sProdCodeAX5000 									:= 		F_ConvProductCodeToString(stSlaveIdentityAX5000);
//Get last 4 characters of the string
sProdCodeAX5000_End4 								:= 		RIGHT(sProdCodeAX5000, 4) ;
//Convert last 4 characters to a number
g_iHMI_ProdCodeAX5000 								:= 		STRING_TO_INT(sProdCodeAX5000_End4);

//In this function block the CRC counts for the individual counts can be decoded
fbAX5000_EcGetSlaveCrcErrorEx(	
							sNetId					:= 		gc_sADSNetID,
							nSlaveAddr				:= 		gc_uiAX5206_EtherCATAdr,
							bExecute				:= 		xExecute,
							tTimeout				:= 		T#2S,
							bBusy					=> 		xAX5000GetSlaveCrc_Busy,
							bError					=> 		xAX5000GetSlaveCrc_Error,
							nErrId					=> 		udiAX5000GetSlaveCrc_ErrId,
							crcError				=> 		g_stHMI_AX5000CrcErrorEx );

//Working Counter: Should remain Zero, If value=1 then data is bad from this device
g_xAX5000_Wc ;


//Get the STATE of the AX5805 terminal and display as a text string
g_sHMI_StateAX5805 									:= 		F_ConvStateToString(g_wStateAX5805);

// slave device's STATE BITS  
g_stHMI_AX5805EcSlaveStateBits 						:=  	F_ConvSlaveStateToBits(g_stAX5805EcSlaveState);

fbAX5805_EcGetSlaveIdentity(		
							sNetId					:= 		gc_sADSNetID,
							nSlaveAddr				:= 		gc_uiAX5805_EtherCATAdr,
							bExecute				:= 		xExecute,
							tTimeout				:= 		T#2S,
							bBusy					=> 		xAX5805SlaveIdentity_Busy,
							bError					=> 		xAX5805SlaveIdentity_Error,
							nErrId					=> 		udiAX5805SlaveIdentity_ErrId,
							identity				=> 		stSlaveIdentityAX5805 );

sProdCodeAX5805 									:= 		F_ConvProductCodeToString(stSlaveIdentityAX5805);
//Get last 4 characters of the string
sProdCodeAX5805_End4 								:= 		RIGHT(sProdCodeAX5805, 4) ;
//Convert last 4 characters to a number
g_iHMI_ProdCodeAX5805 								:= 		STRING_TO_INT(sProdCodeAX5805_End4);

//In this function block the CRC counts for the individual counts can be decoded
fbAX5805_EcGetSlaveCrcErrorEx(	
							sNetId					:= 		gc_sADSNetID,
							nSlaveAddr				:= 		gc_uiAX5805_EtherCATAdr,
							bExecute				:= 		xExecute,
							tTimeout				:= 		T#2S,
							bBusy					=> 		xAX5805GetSlaveCrc_Busy,
							bError					=> 		xAX5805GetSlaveCrc_Error,
							nErrId					=> 		udiAX5805GetSlaveCrc_ErrId,
							crcError				=> 		g_stHMI_AX5805CrcErrorEx );

//Working Counter: Should remain Zero, If value=1 then data is bad from this device
g_xAX5805_Wc ;


//Get the STATE of the EP1908-0002 module and display as a text string
g_sHMI_StateEP1908 									:= 		F_ConvStateToString(g_wStateEP1908);

// slave device's STATE BITS  
g_stHMI_EP1908EcSlaveStateBits 						:=  	F_ConvSlaveStateToBits(g_stEP1908EcSlaveState);

fbEP1908_EcGetSlaveIdentity(		
							sNetId					:= 		gc_sADSNetID,
							nSlaveAddr				:= 		gc_uiEP1908_EtherCATAdr,
							bExecute				:= 		xExecute,
							tTimeout				:= 		T#2S,
							bBusy					=> 		xEP1908SlaveIdentity_Busy,
							bError					=> 		xEP1908SlaveIdentity_Error,
							nErrId					=> 		udiEP1908SlaveIdentity_ErrId,
							identity				=> 		stSlaveIdentityEP1908 );

sProdCodeEP1908 									:= 		F_ConvProductCodeToString(stSlaveIdentityEP1908);
//Get last 4 characters of the string
sProdCodeEP1908_End4 								:= 		RIGHT(sProdCodeEP1908, 4) ;
//Convert last 4 characters to a number
g_iHMI_ProdCodeEP1908 								:= 		STRING_TO_INT(sProdCodeEP1908_End4);

//In this function block the CRC counts for the individual counts can be decoded
fbEP1908_EcGetSlaveCrcErrorEx(	
							sNetId					:= 		gc_sADSNetID,
							nSlaveAddr				:= 		gc_uiEP1908_EtherCATAdr,
							bExecute				:= 		xExecute,
							tTimeout				:= 		T#2S,
							bBusy					=> 		xEP1908GetSlaveCrc_Busy,
							bError					=> 		xEP1908GetSlaveCrc_Error,
							nErrId					=> 		udiEP1908GetSlaveCrc_ErrId,
							crcError				=> 		g_stHMI_EP1908CrcErrorEx );

//Working Counter: Should remain Zero, If value=1 then data is bad from this device
g_xEP1908_Wc ;

*)

//END_IF ;

END_PROGRAM

// ---- POUs/Control_System_Diagnostics/System_Functions.TcPOU
PROGRAM System_Functions
//		8-2-2012
// 		This Program has been supplied by Beckhoff Automation As-Is and is intended only as an example 
//		implementation. Functionality is not guaranteed. 
//
VAR
	//General timer for periodic reads
	T1									:		TON ;
	xExecute							:		BOOL ;
	tTime1								:		TIME ;

	//Get Device Identification
	fbGetDeviceIdentificationEx			:		FB_GetDeviceIdentificationEx ;
	xGetDeviceId_Busy					:		BOOL ;
	xGetDeviceId_Error					:		BOOL ;
	udiGetDeviceId_ErrId				:		UDINT ;
	stDevIdent							:		ST_DeviceIdentificationEx ;

	//Get ADS Router Info
	fbGetRouterStatusInfo				:		FB_GetRouterStatusInfo ;
	xGetRouterStatusInfo_Busy			:		BOOL ;
	xGetRouterStatusInfo_Error			:		BOOL ;
	udiGetRouterStatusInfo_ErrId		:		UDINT ;
	stRouterStatusInfo					:		ST_TcRouterStatusInfo ;


(*
(* Get CPU Usage Info  *)
	fbTC_CpuUsage: TC_CpuUsage;
	bCpuUsage_Busy: BOOL;
	bCpuUsage_Error: BOOL;
	nCpuUsage_ErrId: UDINT;
	nCpuUsage: UDINT;
	nCpuUsage_HMI: UDINT;

(* Get System Latency Values *)
	fbTC_SysLatency: TC_SysLatency;
	bSysLatency_Busy: BOOL;
	bSysLatency_Error: BOOL;
	nSysLatency_ErrId: UDINT;
	nSysLatency_Actual: UDINT;
	nSysLatency_Max: UDINT;
	nSysLatency_Actual_HMI: UDINT;
	nSysLatency_Max_HMI: UDINT;

(* SystemTaskInfoArr[1].cycleTime is in 100ns increments - needed to convert to ms for display*)
	nCycleTime_HMI: LREAL;

(* SystemTaskInfoArr[1].lastExecTime is in 100ns increments - needed to convert to ms for display*)
	nLastExecTime_HMI: LREAL;
	fbGetDeviceIdentificationEx: FB_GetDeviceIdentificationEx;
*)
	fbFB_MDP_ScanModules				: 		FB_MDP_ScanModules;
	eMDP_ModType						: 		E_MDP_ModuleType;
	usiModIdx							: 		USINT;
	xMDP_ScanModules_busy				: 		BOOL;
	xMDP_ScanModules_Error				: 		BOOL;
	udiMDP_ScanModules_ErrID			: 		UDINT;
	bMDP_ScanModules_DynModID			: 		BYTE;
	usiMDP_ScanModules_ModTypCnt		: 		USINT;
	usiMDP_ScanModules_ModCnt			: 		USINT;

	fbFB_MDP_ReadModuleContent 			:		FB_MDP_ReadModuleContent ;
	ST_MDP_Addr 						:		ST_MDP_Addr ;
	dwMB_Buffer							: 		DWORD ;
	xMDP_Motherboard_ReadModContent_Busy: 		BOOL ;
	xMDP_Motherboard_ReadModContent_Error: 		BOOL ;
	udiMDP_Motherboard_ReadModContent_ErrID: 	UDINT ;
	usiMDP_Motherboard_ReadModContent_ErrPOS: 	USINT ;
	arrMDP_Motherboard_StartIdx			: 		ARRAY [0..255] OF UINT ;

	fbFB_MDP_SplitErrorID				: 		FB_MDP_SplitErrorID ;
	eMDP_ErrGroup 						:		E_MDP_ErrGroup ;
	uiMDP_Motherboard_ReadModContent_ErrCODE:	UINT ;

	fbFB_MDP_ReadModuleHeader			: 		FB_MDP_ReadModuleHeader ;
	xMDP_Motherboard_ReadModHeader_Busy	: 		BOOL ;
	xMDP_Motherboard_ReadModHeader_Error: 		BOOL ;
	udiMDP_Motherboard_ReadModHeader_ErrID: 	UDINT ;
	ST_MDP_Motherboard_ReadModHeader 	:		ST_MDP_ModuleHeader ;

	fbFB_MDP_CPU_Read1					: 		FB_MDP_CPU_Read;
	ST_CPUModHdr 						:		ST_MDP_ModuleHeader ;
	ST_CPUModContent 					: 		ST_MDP_CPU ;

	fbFB_MDP_Mainboard_ReadTBL1			: 		FB_MDP_Mainboard_ReadTBL1;
	ST_MainboardModHdrTBL1				:		ST_MDP_ModuleHeader ;
	ST_MainboardModContentTBL1			: 		ST_MDP_MainboardTBL1 ;

	fbFB_MDP_Mainboard_ReadTBL2			: 		FB_MDP_Mainboard_ReadTBL2 ;
	ST_MainboardModHdrTBL2				:		ST_MDP_ModuleHeader ;
	ST_MainboardModContentTBL2			: 		ST_MDP_MainboardTBL2 ;

	fbFB_MDP_Mainboard_ReadTBL3			: 		FB_MDP_Mainboard_ReadTBL3 ;
	ST_MainboardModHdrTBL3				:		ST_MDP_ModuleHeader ;
	ST_MainboardModContentTBL3			: 		ST_MDP_MainboardTBL3 ;

	fbFB_MDP_Mainboard_ReadTBL4			: 		FB_MDP_Mainboard_ReadTBL4 ;
	ST_MainboardModHdrTBL4				:		ST_MDP_ModuleHeader ;
	ST_MainboardModContentTBL4			: 		ST_MDP_MainboardTBL4 ;
	
	fbFB_MDP_NIC0_Read					: 		FB_MDP_NIC_Read ;
	ST_NIC0_ModHdr						: 		ST_MDP_ModuleHeader ;
	ST_NIC0_ModContent					: 		ST_MDP_NIC_Properties ;
	
	fbFB_MDP_NIC1_Read					: 		FB_MDP_NIC_Read ;
	ST_NIC1_ModHdr						: 		ST_MDP_ModuleHeader ;
	ST_NIC1_ModContent					: 		ST_MDP_NIC_Properties ;	
	lrOperTimeHrs						: 		LREAL ;
	lrOperTimeDays						: 		LREAL ;
	lrOperTimeYears						: 		LREAL ;

	fbFB_MDP_Time1_Read					: 		FB_MDP_Time_ReadTBL1 ;
	ST_Time1_ModHdr						: 		ST_MDP_ModuleHeader ;
	ST_Time1_ModContent					: 		ST_MDP_TimeTBL1 ;
END_VAR

//		8-2-2012
// 		This Program has been supplied by Beckhoff Automation As-Is and is intended only as an example 
//		implementation. Functionality is not guaranteed. 
//

//IF g_bHMI_ScreenBeingDisplayed = 90 THEN
//Create the xExecute bit for continuous timed interval FB calls
T1(IN:= NOT xExecute, PT:= T#2S, Q=> xExecute, ET=>tTime1 );

(* Computer/Controller Device Info - Get CX and TwinCAT version info
   from the resulting structure "stDevIdent" - display only when the 
   function block is not BUSY retrieving the data else the display
   will "blink" because while the FB is BUSY the values go to 0 or
   "blank" text *)
fbGetDeviceIdentificationEx(
							bExecute					:= 		xExecute, 
							tTimeout					:= 		T#2S, 
							sNetId						:= 		'', 
							bBusy						=> 		xGetDeviceId_Busy, 
							bError						=> 		xGetDeviceId_Error, 
							nErrorID					=> 		udiGetDeviceId_ErrId, 
							stDevIdent					=> 		stDevIdent );
							
IF NOT xGetDeviceId_Busy THEN 
							g_stHMI_DevIdent 			:= 		stDevIdent ; 
END_IF ;

g_stHMI_AppInfo 										:= _AppInfo  ;

//ADS Router Status info
fbGetRouterStatusInfo(		
							sNetId						:= 		'',
							bExecute					:= 		xExecute,
							tTimeout					:= 		T#2S,
							bBusy						=> 		xGetRouterStatusInfo_Busy,
							bError						=> 		xGetRouterStatusInfo_Error,
							nErrID						=> 		udiGetRouterStatusInfo_ErrId,
							info						=> 		stRouterStatusInfo );
							
IF NOT xGetRouterStatusInfo_Busy THEN 
							g_stHMI_RouterStatusInfo	:= 		stRouterStatusInfo ; 
END_IF ;

g_stHMI_PlcTaskSystemInfo 								:= 		_TaskInfo[_AppInfo.TaskCnt] ;
g_lrHMI_PlcTaskSystemInfo_CycleTime 					:= 		g_stHMI_PlcTaskSystemInfo.CycleTime / 10.0 ;
g_lrHMI_PlcTaskSystemInfo_LastExecTime 					:= 		g_stHMI_PlcTaskSystemInfo.LastExecTime / 10.0 ;

//In order to be able to query or set an MDP parameter, the Dynamic Module ID of 
//the module in which the parameter is located must be known.
fbFB_MDP_ScanModules(
							bExecute					:= 		xExecute, 
							nModuleType					:= 		eMDP_ModType, 
							iModIdx						:= 		usiModIdx, 
							tTimeout					:= 		T#2S, 
							sAmsNetId					:= 		'', 
							bBusy						=> 		xMDP_ScanModules_busy, 
							bError						=> 		xMDP_ScanModules_Error, 
							nErrID						=> 		udiMDP_ScanModules_ErrID, 
							nDynModuleId				=> 		bMDP_ScanModules_DynModID, 
							iModuleTypeCount			=> 		usiMDP_ScanModules_ModTypCnt, 
							iModuleCount				=> 		usiMDP_ScanModules_ModCnt );

// The function block enables the header of an MDP module to be queried
fbFB_MDP_ReadModuleHeader(
							bExecute					:= 		xExecute, 
							nDynModuleId				:= 		4, 
							tTimeout					:= 		T#2S, 
							sAmsNetId					:= 		'', 
							bBusy						=> 		xMDP_Motherboard_ReadModHeader_Busy, 
							bError						=> 		xMDP_Motherboard_ReadModHeader_Error, 
							nErrID						=> 		udiMDP_Motherboard_ReadModHeader_ErrID, 
							stMDP_ModHeader				=> 		ST_MDP_Motherboard_ReadModHeader);							
							

fbFB_MDP_CPU_Read1(
							xExecute					:= 		xExecute, 
							tTimeout					:= 		T#2S, 
							usiModIdx					:= 		0, 
							sAmsNetId					:= 		'', 
							bBusy						=> 		, 
							bError						=> 		, 
							nErrID						=> 		, 
							iErrPos						=> 		, 
							stMDP_ModuleHeader			=> 		ST_CPUModHdr, 
							stMDP_ModuleContent			=> 		ST_CPUModContent);							

g_lrHMI_CPUfrequency 									:=		ST_CPUModContent.udiCPUfrequency / 1000.0	; // CPU Clock Frequency in GHz				
g_iHMI_CPUusage											:=		ST_CPUModContent.uiCPUusage ;  // CPU Usage in percent
g_iHMI_CPUtemperature 									:= 		ST_CPUModContent.iCPUtemp ; // CPU Temperature in DegC	

fbFB_MDP_Mainboard_ReadTBL1(
							xExecute					:= 		xExecute, 
							tTimeout					:= 		T#2S, 
							usiModIdx					:= 		0, 
							sAmsNetId					:= 		'', 
							bBusy						=> 		, 
							bError						=> 		, 
							nErrID						=> 		, 
							iErrPos						=> 		, 
							stMDP_ModuleHeader			=> 		ST_MainboardModHdrTBL1, 
							stMDP_ModuleContent			=> 		ST_MainboardModContentTBL1);


g_sHMI_MainboardType 									:= 		ST_MainboardModContentTBL1.sMainboardType ;
g_sHMI_MainboardSN 										:= 		ST_MainboardModContentTBL1.sMainboardSN ;
g_sHMI_MainboardProdDate								:= 		ST_MainboardModContentTBL1.sMainboardProdDate ;
g_udiHMI_MainboardBootCount								:= 		ST_MainboardModContentTBL1.udiMainboardBootCount ;
lrOperTimeHrs											:= 		ST_MainboardModContentTBL1.udiMainboardOperTime / 60.0 ;
lrOperTimeDays											:= 		lrOperTimeHrs / 24.0 ;
g_udiHMI_MainboardOperTimeDays 							:= 		TRUNC(lrOperTimeDays) ;
g_lrHMI_MainboardOperTimeHrs							:=		24.0 * (lrOperTimeDays - UDINT_TO_LREAL(g_udiHMI_MainboardOperTimeDays)) ;
g_diHMI_MainboardMinTemp								:= 		ST_MainboardModContentTBL1.diMainboardMinTemp ;
g_diHMI_MainboardMaxTemp								:= 		ST_MainboardModContentTBL1.diMainboardMaxTemp ;
g_lrHMI_MainboardMinVolt								:= 		ST_MainboardModContentTBL1.diMainboardMinVolt / 1000.0 ;
g_lrHMI_MainboardMaxVolt								:= 		ST_MainboardModContentTBL1.diMainboardMaxVolt / 1000.0 ;
g_iHMI_MainboardActualTemp								:= 		ST_MainboardModContentTBL1.iMainboardActualTemp ;


fbFB_MDP_Mainboard_ReadTBL2(
							xExecute					:= 		xExecute, 
							tTimeout					:= 		T#2S, 
							usiModIdx						:= 		0, 
							sAmsNetId					:= 		'', 
							bBusy						=> 		, 
							bError						=> 		, 
							nErrID						=> 		, 
							iErrPos						=> 		, 
							stMDP_ModuleHeader			=> 		ST_MainboardModHdrTBL2, 
							stMDP_ModuleContent			=> 		ST_MainboardModContentTBL2);


g_bHMI_MainboardRevision 								:= 		ST_MainboardModContentTBL2.usiMainboardRevision ;
g_bHMI_MainboardBiosMajVers 							:= 		ST_MainboardModContentTBL2.usiMainboardBiosMajVers ;
g_bHMI_MainboardBiosMinVers 							:= 		ST_MainboardModContentTBL2.usiMainboardBiosMinVers ;


fbFB_MDP_Mainboard_ReadTBL3(
							xExecute					:= 		xExecute, 
							tTimeout					:= 		T#2S, 
							usiModIdx						:= 		0, 
							sAmsNetId					:= 		'', 
							bBusy						=> 		, 
							bError						=> 		, 
							nErrID						=> 		, 
							iErrPos						=> 		, 
							stMDP_ModuleHeader			=> 		ST_MainboardModHdrTBL3, 
							stMDP_ModuleContent			=> 		ST_MainboardModContentTBL3);							

g_sHMI_Mainboard1p05v 									:= 		ST_MainboardModContentTBL3.sMainboard1p05v ;
g_sHMI_MainboardVccCore 								:= 		ST_MainboardModContentTBL3.sMainboardVccCore ;
g_sHMI_Mainboard5v 										:= 		ST_MainboardModContentTBL3.sMainboard5v ;
g_sHMI_Mainboard12v 									:= 		ST_MainboardModContentTBL3.sMainboard12v ;
g_sHMI_MainboardVBatt 									:= 		ST_MainboardModContentTBL3.sMainboardVBatt ;
g_sHMI_MainboardPwrCtrlVcc 								:= 		ST_MainboardModContentTBL3.sMainboardPwrCtrlVcc ;
g_sHMI_MainboardCX2100_5v 								:= 		ST_MainboardModContentTBL3.sMainboardCX2100_5v ;
g_sHMI_MainboardCX2100_12v 								:= 		ST_MainboardModContentTBL3.sMainboardCX2100_12v ;
g_sHMI_MainboardCX2100_24v 								:= 		ST_MainboardModContentTBL3.sMainboardCX2100_24v ;

					
fbFB_MDP_Mainboard_ReadTBL4(
							xExecute					:= 		xExecute, 
							tTimeout					:= 		T#2S, 
							usiModIdx						:= 		0, 
							sAmsNetId					:= 		'', 
							bBusy						=> 		, 
							bError						=> 		, 
							nErrID						=> 		, 
							iErrPos						=> 		, 
							stMDP_ModuleHeader			=> 		ST_MainboardModHdrTBL4, 
							stMDP_ModuleContent			=> 		ST_MainboardModContentTBL4);

g_lrHMI_Mainboard1p05v 									:= 		ST_MainboardModContentTBL4.iMainboard1p05v / 1000.0 ;
g_lrHMI_MainboardVccCore 								:= 		ST_MainboardModContentTBL4.iMainboardVccCore / 1000.0 ;
g_lrHMI_Mainboard5v 									:= 		ST_MainboardModContentTBL4.iMainboard5v / 1000.0 ;
g_lrHMI_Mainboard12v 									:= 		ST_MainboardModContentTBL4.iMainboard12v / 1000.0 ;
g_lrHMI_MainboardVBatt 									:= 		ST_MainboardModContentTBL4.iMainboardVBatt / 1000.0 ;
g_lrHMI_MainboardPwrCtrlVcc 							:= 		ST_MainboardModContentTBL4.iMainboardPwrCtrlVcc / 1000.0 ;
g_lrHMI_MainboardCX2100_5v 								:= 		ST_MainboardModContentTBL4.iMainboardCX2100_5v / 1000.0 ;
g_lrHMI_MainboardCX2100_12v 							:= 		ST_MainboardModContentTBL4.iMainboardCX2100_12v / 1000.0 ;
g_lrHMI_MainboardCX2100_24v 							:= 		ST_MainboardModContentTBL4.iMainboardCX2100_24v / 1000.0 ; 


fbFB_MDP_NIC0_Read(
							xExecute					:= 		xExecute, 
							tTimeout					:= 		T#2S, 
							usiModIdx					:= 		0, 
							sAmsNetId					:= 		'', 
							bBusy						=> 		, 
							bError						=> 		, 
							nErrID						=> 		, 
							iErrPos						=> 		, 
							stMDP_ModuleHeader			=> 		ST_NIC0_ModHdr, 
							stMDP_ModuleContent			=> 		ST_NIC0_ModContent);

fbFB_MDP_NIC1_Read(
							xExecute					:= 		xExecute, 
							tTimeout					:= 		T#2S, 
							usiModIdx					:= 		1, 
							sAmsNetId					:= 		'', 
							bBusy						=> 		, 
							bError						=> 		, 
							nErrID						=> 		, 
							iErrPos						=> 		, 
							stMDP_ModuleHeader			=> 		ST_NIC1_ModHdr, 
							stMDP_ModuleContent			=> 		ST_NIC1_ModContent);

fbFB_MDP_Time1_Read(
							xExecute					:= 		xExecute, 
							tTimeout					:= 		T#2S, 
							usiModIdx					:= 		0, 
							sAmsNetId					:= 		'', 
							bBusy						=> 		, 
							bError						=> 		, 
							nErrID						=> 		, 
							iErrPos						=> 		, 
							stMDP_ModuleHeader			=> 		ST_Time1_ModHdr, 
							stMDP_ModuleContent			=> 		ST_Time1_ModContent);				
//	END_IF ;

END_PROGRAM

// ---- POUs/MDP_Function_Blocks/FB_MDP_Mainboard_ReadTBL1.TcPOU
FUNCTION_BLOCK FB_MDP_Mainboard_ReadTBL1

VAR_INPUT
	xExecute				: BOOL;								// Function block execution is triggered by a rising edge at this input
	tTimeout				: TIME		:= DEFAULT_ADS_TIMEOUT;	// States the time before the function is cancelled
	usiModIdx				: USINT		:= 0;					// Index number of chosen MDP device
	sAmsNetId				: T_AmsNetId;						// keep empty '' for the local device
END_VAR

VAR_OUTPUT
	xBusy					: BOOL;
	xError					: BOOL;
	udiErrID				: UDINT;
	usiErrPos				: USINT;							// If a subindex is not supported, iErrPos indicates at which subindex the error appears first
	stMDP_ModuleHeader		: ST_MDP_ModuleHeader;
	stMDP_ModuleContent		: ST_MDP_MainboardTBL1;	
END_VAR

VAR
	fbMDP_ReadModule		: FB_MDP_ReadModule;
	arrData					: ARRAY[0..60] OF BYTE;				// requested data
	arrStartIdx				: ARRAY[0..15] OF UINT;				// startindexes in bytes of each subindex element

	stMDP_Addr				: ST_MDP_Addr;
	eModuleType				: E_MDP_ModuleType;
	usiSubIdxCount			: USINT;

	xSubExecute				: BOOL;
	xReadBusy				: BOOL;

	RisingEdge				: R_TRIG;
	TimeOut					: TON;								// general timeout	
END_VAR

RisingEdge( CLK					:= xExecute );
IF NOT xBusy THEN										// FB only react to the external execute if it is not busy
	IF RisingEdge.Q THEN
		xBusy					:= TRUE;

		// reset variables
		xError					:= FALSE;
		udiErrID				:= 0;
		usiErrPos				:= 0;
		xSubExecute				:= TRUE;

		// specific values for Mainboard content
		stMDP_Addr.nArea		:= 16#08;
//		stMDP_Addr.nModuleId;							will be allocated dynamically
		stMDP_Addr.nTableId		:= 16#01;
//		stMDP_Addr.nFlag;								not used up to now
//		stMDP_Addr.nSubIdx;								all subindexes will be requested
		eModuleType				:= eMDP_ModT_Mainboard;
		usiSubIdxCount			:= 11;					// TableId 16#01 contains 10 elements

		MEMSET( ADR(arrData), 0, SIZEOF(arrData) );		// reset buffer

		TimeOut(IN 				:= FALSE);
		TimeOut(PT 				:= tTimeout, IN 	:= TRUE);
	END_IF
END_IF


IF xBusy THEN
	IF xSubExecute THEN
		xSubExecute 			:= FALSE;

		fbMDP_ReadModule( bExecute := FALSE );
		fbMDP_ReadModule(
			stMDP_Addr			:= stMDP_Addr,
			eModuleType			:= eModuleType,
			iModIdx				:= usiModIdx,
			iSubIdxCount		:= usiSubIdxCount,
			bExecute			:= TRUE,
			tTimeout			:= tTimeout,
			pDstBuf				:= ADR(arrData),
			cbDstBufLen			:= SIZEOF(arrData),
			sAmsNetId			:= sAmsNetId,

			bBusy				=> xReadBusy,
			bError				=> xError,
			nErrID				=> udiErrID,
			iErrPos				=> usiErrPos,
			stMDP_DynAddr		=> ,
			iModuleTypeCount	=> ,
			iModuleCount		=> ,
			stMDP_ModuleHeader	=> ,
			arrStartIdx			=> ,
		);
	ELSE
		fbMDP_ReadModule(
			bExecute			:= FALSE,

			bBusy				=> xReadBusy,
			bError				=> xError,
			nErrID 				=> udiErrID,
			iErrPos				=> usiErrPos,
		 );
		IF NOT xReadBusy THEN
			// allocate received module header
			stMDP_ModuleHeader	:= fbMDP_ReadModule.stMDP_ModuleHeader;
			// allocate information of startindexes in data buffer
			MEMCPY(ADR(arrStartIdx), ADR(fbMDP_ReadModule.arrStartIdx), SIZEOF(arrStartIdx) );
			// reset module content struct
			MEMSET( ADR(stMDP_ModuleContent), 0, SIZEOF(stMDP_ModuleContent) );
			// allocate received data to NIC struct
			stMDP_ModuleContent.uiLen		:= arrData[0];
			MEMCPY(ADR(stMDP_ModuleContent.sMainboardType),			ADR(arrData)+arrStartIdx[1],	MIN(arrStartIdx[2]-arrStartIdx[1],	SIZEOF(stMDP_ModuleContent.sMainboardType))     );
			MEMCPY(ADR(stMDP_ModuleContent.sMainboardSN),			ADR(arrData)+arrStartIdx[2],	MIN(arrStartIdx[3]-arrStartIdx[2],	SIZEOF(stMDP_ModuleContent.sMainboardSN))     );
			MEMCPY(ADR(stMDP_ModuleContent.sMainboardProdDate),		ADR(arrData)+arrStartIdx[3],	MIN(arrStartIdx[4]-arrStartIdx[3],	SIZEOF(stMDP_ModuleContent.sMainboardProdDate))     );
			MEMCPY(ADR(stMDP_ModuleContent.udiMainboardBootCount),	ADR(arrData)+arrStartIdx[4],	MIN(arrStartIdx[5]-arrStartIdx[4],	SIZEOF(stMDP_ModuleContent.udiMainboardBootCount))     );
			MEMCPY(ADR(stMDP_ModuleContent.udiMainboardOperTime),	ADR(arrData)+arrStartIdx[5],	MIN(arrStartIdx[6]-arrStartIdx[5],	SIZEOF(stMDP_ModuleContent.udiMainboardOperTime))     );
			MEMCPY(ADR(stMDP_ModuleContent.diMainboardMinTemp),		ADR(arrData)+arrStartIdx[6],	MIN(arrStartIdx[7]-arrStartIdx[6],	SIZEOF(stMDP_ModuleContent.diMainboardMinTemp))     );
			MEMCPY(ADR(stMDP_ModuleContent.diMainboardMaxTemp),		ADR(arrData)+arrStartIdx[7],	MIN(arrStartIdx[8]-arrStartIdx[7],	SIZEOF(stMDP_ModuleContent.diMainboardMaxTemp))     );
			MEMCPY(ADR(stMDP_ModuleContent.diMainboardMinVolt),		ADR(arrData)+arrStartIdx[8],	MIN(arrStartIdx[9]-arrStartIdx[8],	SIZEOF(stMDP_ModuleContent.diMainboardMinVolt))     );
			MEMCPY(ADR(stMDP_ModuleContent.diMainboardMaxVolt),		ADR(arrData)+arrStartIdx[9],	MIN(arrStartIdx[10]-arrStartIdx[9],	SIZEOF(stMDP_ModuleContent.diMainboardMaxVolt))     );
			MEMCPY(ADR(stMDP_ModuleContent.iMainboardActualTemp),	ADR(arrData)+arrStartIdx[10],	MIN(arrStartIdx[11]-arrStartIdx[10],SIZEOF(stMDP_ModuleContent.iMainboardActualTemp))     );

			// reset FB
			xBusy 				:= FALSE;
		END_IF
	END_IF

	// check timeout
	TimeOut();
	IF TimeOut.Q THEN
		TimeOut(IN 				:= FALSE);
		xError					:= TRUE;
		udiErrID				:= INT_TO_UINT(eMDP_Err_PLC) * 16#10000 + INT_TO_UINT(eMDP_ErrPLC_TimeOut);
	END_IF
END_IF

IF xError THEN
	// reset FB
	xBusy 						:= FALSE;
END_IF

END_FUNCTION_BLOCK

// ---- POUs/MDP_Function_Blocks/FB_MDP_NIC_Read.TcPOU
FUNCTION_BLOCK FB_MDP_NIC_Read
VAR_INPUT
	xExecute			: BOOL;								// Function block execution is triggered by a rising edge at this input
	tTimeout			: TIME		:= DEFAULT_ADS_TIMEOUT;	// States the time before the function is cancelled
	usiModIdx			: USINT		:= 0;					// Index number of chosen MDP device
	sAmsNetId			: T_AmsNetId;						// keep empty '' for the local device	
END_VAR
VAR_OUTPUT
	xBusy				: BOOL;
	xError				: BOOL;
	udiErrID			: UDINT;
	usiErrPos			: USINT;							// If a subindex is not supported, iErrPos indicates at which subindex the error appears first
	stMDP_ModuleHeader	: ST_MDP_ModuleHeader;
	stMDP_ModuleContent	: ST_MDP_NIC_Properties;	
END_VAR
VAR
	fbMDP_ReadModule	: FB_MDP_ReadModule;
	arrData				: ARRAY[0..799] OF BYTE;			// requested data
	arrStartIdx			: ARRAY[0..255] OF UINT;			// startindexes in bytes of each subindex element

	stMDP_Addr			: ST_MDP_Addr;
	eModuleType			: E_MDP_ModuleType;
	usiSubIdxCount		: USINT;

	xSubExecute			: BOOL;
	xReadBusy			: BOOL;

	RisingEdge			: R_TRIG;
	TimeOut				: TON;								// general timeout
END_VAR

RisingEdge( CLK					:= xExecute );
IF NOT xBusy THEN											// FB only react to the external execute if it is not busy
	IF RisingEdge.Q THEN
		xBusy					:= TRUE;
		
		// reset variables
		xError					:= FALSE;
		udiErrID				:= 0;
		usiErrPos				:= 0;
		xSubExecute				:= TRUE;
	
		// specific values for NIC content
		stMDP_Addr.nArea		:= 16#08;
//		stMDP_Addr.nModuleId;								will be allocated dynamically
		stMDP_Addr.nTableId		:= 16#01;
//		stMDP_Addr.nFlag;									not used up to now
//		stMDP_Addr.nSubIdx;									all subindexes will be requested
		eModuleType				:= eMDP_ModT_NIC;
		usiSubIdxCount			:= 6;						// TableId 16#01 contains 6 elements

		MEMSET( ADR(arrData), 0, SIZEOF(arrData) );			// reset buffer

		TimeOut(IN 				:= FALSE);
		TimeOut(PT 				:= tTimeout, IN := TRUE);
	END_IF
END_IF


IF xBusy THEN
	IF xSubExecute THEN
		xSubExecute 			:= FALSE;

		fbMDP_ReadModule( bExecute := FALSE );
		fbMDP_ReadModule(
			stMDP_Addr			:= stMDP_Addr,
			eModuleType			:= eModuleType,
			iModIdx				:= usiModIdx,
			iSubIdxCount		:= usiSubIdxCount,
			bExecute			:= TRUE,
			tTimeout			:= tTimeout,
			pDstBuf				:= ADR(arrData),
			cbDstBufLen			:= SIZEOF(arrData),
			sAmsNetId			:= sAmsNetId,

			bBusy				=> xReadBusy,
			bError				=> xError,
			nErrID				=> udiErrID,
			iErrPos				=> usiErrPos,
			stMDP_DynAddr		=> ,
			iModuleTypeCount	=> ,
			iModuleCount		=> ,
			stMDP_ModuleHeader	=> ,
			arrStartIdx			=> ,
		);
	ELSE
		fbMDP_ReadModule(
			bExecute			:= FALSE,

			bBusy				=> xReadBusy,
			bError				=> xError,
			nErrID 				=> udiErrID,
			iErrPos				=> usiErrPos,
		);
		IF NOT xReadBusy THEN
			// allocate received module header
			stMDP_ModuleHeader	:= fbMDP_ReadModule.stMDP_ModuleHeader;
			// allocate information of startindexes in data buffer
			MEMCPY(ADR(arrStartIdx), ADR(fbMDP_ReadModule.arrStartIdx), SIZEOF(arrStartIdx) );
			// reset module content struct
			MEMSET( ADR(stMDP_ModuleContent), 0, SIZEOF(stMDP_ModuleContent) );
			// allocate received data to NIC struct
			stMDP_ModuleContent.uiLen		:= arrData[0];
			MEMCPY(ADR(stMDP_ModuleContent.sMACAddress), 	ADR(arrData)+arrStartIdx[1], MIN(arrStartIdx[2]-arrStartIdx[1], SIZEOF(stMDP_ModuleContent.sMACAddress)) );
			MEMCPY(ADR(stMDP_ModuleContent.sIPAddress), 	ADR(arrData)+arrStartIdx[2], MIN(arrStartIdx[3]-arrStartIdx[2], SIZEOF(stMDP_ModuleContent.sIPAddress))  );
			MEMCPY(ADR(stMDP_ModuleContent.sSubnetMask), 	ADR(arrData)+arrStartIdx[3], MIN(arrStartIdx[4]-arrStartIdx[3], SIZEOF(stMDP_ModuleContent.sSubnetMask)) );
			MEMCPY(ADR(stMDP_ModuleContent.xDHCP), 			ADR(arrData)+arrStartIdx[4], 1);
			MEMCPY(ADR(stMDP_ModuleContent.sDefaultGateway),ADR(arrData)+arrStartIdx[5], MIN(arrStartIdx[6]-arrStartIdx[5], SIZEOF(stMDP_ModuleContent.sDefaultGateway)) );

			// reset FB
			xBusy 				:= FALSE;
		END_IF
	END_IF

	// check timeout
	TimeOut();
	IF TimeOut.Q THEN
		TimeOut(IN 				:= FALSE);
		xError					:= TRUE;
		udiErrID				:= INT_TO_UINT(eMDP_Err_PLC) * 16#10000 + INT_TO_UINT(eMDP_ErrPLC_TimeOut);
	END_IF
END_IF

IF xError THEN
	// reset FB
	xBusy 						:= FALSE;
END_IF

END_FUNCTION_BLOCK

// ---- POUs/MDP_Function_Blocks/FB_MDP_Time_ReadTBL1.TcPOU
FUNCTION_BLOCK FB_MDP_Time_ReadTBL1

VAR_INPUT
	xExecute				: BOOL;								// Function block execution is triggered by a rising edge at this input
	tTimeout				: TIME		:= DEFAULT_ADS_TIMEOUT;	// States the time before the function is cancelled
	usiModIdx				: USINT		:= 0;					// Index number of chosen MDP device
	sAmsNetId				: T_AmsNetId;						// keep empty '' for the local device
END_VAR

VAR_OUTPUT
	xBusy					: BOOL;
	xError					: BOOL;
	udiErrID				: UDINT;
	usiErrPos				: USINT;							// If a subindex is not supported, iErrPos indicates at which subindex the error appears first
	stMDP_ModuleHeader		: ST_MDP_ModuleHeader;
	stMDP_ModuleContent		: ST_MDP_TimeTBL1;	
END_VAR

VAR
	fbMDP_ReadModule		: FB_MDP_ReadModule;
	arrData					: ARRAY[0..40] OF BYTE;				// requested data
	arrStartIdx				: ARRAY[0..6] OF UINT;				// startindexes in bytes of each subindex element

	stMDP_Addr				: ST_MDP_Addr;
	eModuleType				: E_MDP_ModuleType;
	usiSubIdxCount			: USINT;

	xSubExecute				: BOOL;
	xReadBusy				: BOOL;

	RisingEdge				: R_TRIG;
	TimeOut					: TON;								// general timeout	
END_VAR

RisingEdge( CLK					:= xExecute );
IF NOT xBusy THEN										// FB only react to the external execute if it is not busy
	IF RisingEdge.Q THEN
		xBusy					:= TRUE;

		// reset variables
		xError					:= FALSE;
		udiErrID				:= 0;
		usiErrPos				:= 0;
		xSubExecute				:= TRUE;

		// specific values for Mainboard content
		stMDP_Addr.nArea		:= 16#08;
//		stMDP_Addr.nModuleId;							will be allocated dynamically
		stMDP_Addr.nTableId		:= 16#01;
//		stMDP_Addr.nFlag;								not used up to now
//		stMDP_Addr.nSubIdx;								all subindexes will be requested
		eModuleType				:= eMDP_ModT_Time;
		usiSubIdxCount			:= 6;					// TableId 16#01 contains 5 elements

		MEMSET( ADR(arrData), 0, SIZEOF(arrData) );		// reset buffer

		TimeOut(IN 				:= FALSE);
		TimeOut(PT 				:= tTimeout, IN 	:= TRUE);
	END_IF
END_IF


IF xBusy THEN
	IF xSubExecute THEN
		xSubExecute 			:= FALSE;

		fbMDP_ReadModule( bExecute := FALSE );
		fbMDP_ReadModule(
			stMDP_Addr			:= stMDP_Addr,
			eModuleType			:= eModuleType,
			iModIdx				:= usiModIdx,
			iSubIdxCount		:= usiSubIdxCount,
			bExecute			:= TRUE,
			tTimeout			:= tTimeout,
			pDstBuf				:= ADR(arrData),
			cbDstBufLen			:= SIZEOF(arrData),
			sAmsNetId			:= sAmsNetId,

			bBusy				=> xReadBusy,
			bError				=> xError,
			nErrID				=> udiErrID,
			iErrPos				=> usiErrPos,
			stMDP_DynAddr		=> ,
			iModuleTypeCount	=> ,
			iModuleCount		=> ,
			stMDP_ModuleHeader	=> ,
			arrStartIdx			=> ,
		);
	ELSE
		fbMDP_ReadModule(
			bExecute			:= FALSE,

			bBusy				=> xReadBusy,
			bError				=> xError,
			nErrID 				=> udiErrID,
			iErrPos				=> usiErrPos,
		 );
		IF NOT xReadBusy THEN
			// allocate received module header
			stMDP_ModuleHeader	:= fbMDP_ReadModule.stMDP_ModuleHeader;
			// allocate information of startindexes in data buffer
			MEMCPY(ADR(arrStartIdx), ADR(fbMDP_ReadModule.arrStartIdx), SIZEOF(arrStartIdx) );
			// reset module content struct
			MEMSET( ADR(stMDP_ModuleContent), 0, SIZEOF(stMDP_ModuleContent) );
			// allocate received data to NIC struct
			stMDP_ModuleContent.uiLen		:= arrData[0];
			MEMCPY(ADR(stMDP_ModuleContent.sSNTP_Server),				ADR(arrData)+arrStartIdx[1],	MIN(arrStartIdx[2]-arrStartIdx[1],	SIZEOF(stMDP_ModuleContent.sSNTP_Server))     );
			MEMCPY(ADR(stMDP_ModuleContent.udiSNTP_Refresh),			ADR(arrData)+arrStartIdx[2],	MIN(arrStartIdx[3]-arrStartIdx[2],	SIZEOF(stMDP_ModuleContent.udiSNTP_Refresh))     );
			MEMCPY(ADR(stMDP_ModuleContent.udiSec_Since_1_1_1970),		ADR(arrData)+arrStartIdx[3],	MIN(arrStartIdx[4]-arrStartIdx[3],	SIZEOF(stMDP_ModuleContent.udiSec_Since_1_1_1970))     );
			MEMCPY(ADR(stMDP_ModuleContent.sDateTime_Presentation),		ADR(arrData)+arrStartIdx[4],	MIN(arrStartIdx[5]-arrStartIdx[4],	SIZEOF(stMDP_ModuleContent.sDateTime_Presentation))     );
			MEMCPY(ADR(stMDP_ModuleContent.uiTimezone),					ADR(arrData)+arrStartIdx[5],	MIN(arrStartIdx[6]-arrStartIdx[5],	SIZEOF(stMDP_ModuleContent.uiTimezone))     );

			// reset FB
			xBusy 				:= FALSE;
		END_IF
	END_IF

	// check timeout
	TimeOut();
	IF TimeOut.Q THEN
		TimeOut(IN 				:= FALSE);
		xError					:= TRUE;
		udiErrID				:= INT_TO_UINT(eMDP_Err_PLC) * 16#10000 + INT_TO_UINT(eMDP_ErrPLC_TimeOut);
	END_IF
END_IF

IF xError THEN
	// reset FB
	xBusy 						:= FALSE;
END_IF

END_FUNCTION_BLOCK

// ---- POUs/Safety_Diagnostics/EL6900_ADS_Reads.TcPOU
PROGRAM EL6900_ADS_Reads
//		8-2-2012
// 		This Program has been supplied by Beckhoff Automation As-Is and is intended only as an example 
//		implementation. Functionality is not guaranteed. 
//
VAR
	//Time to check CoE values
	T1							: 		TON ;
	xExecute					: 		BOOL ;
	tTime1						: 		TIME ;

	//Counter for just some very simple sequencing
	C1							: 		CTU ;
	xReset						: 		BOOL ;
	wPreset						: 		WORD := 10 ;
	xDone						: 		BOOL ;
	wCount						: 		WORD ;

	//Read the serial number out of the EL6900
	fbEL6900Sn_ADSRead			: 		ADSREAD ;
	dwEL6900_Sn					: 		DWORD ;
	xEL6900Sn_busy				: 		BOOL ;
	xEL6900Sn_Err				: 		BOOL ;
	xEL6900Sn_ErrID				: 		UDINT ;

	//Read the DIP Switch Setting out of the EL6900
	fbEL6900DSw_ADSRead			: 		ADSREAD ;
	wEL6900_DSw					: 		WORD ;
	xEL6900DSw_busy				: 		BOOL ;
	xEL6900DSw_Err				: 		BOOL ;
	udiEL6900DSw_ErrID			: 		UDINT ;

	//Read the Hardware Version of the EL6900 Logic Terminal
	fbEL6900_HWvers_EcCoESdoRead: 		FB_EcCoESdoRead ;
	sEL6900_HWvers				: 		STRING(2) ;
	xEL6900_HWvers_Busy			: 		BOOL ;
	xEL6900_HWvers_Err			: 		BOOL ;
	udiEL6900_HWvers_ErrID		: 		UDINT ;

	//Read the Software Version of the EL6900 Logic Terminal (It's f/w)
	fbEL6900_FWvers_EcCoESdoRead: 		FB_EcCoESdoRead ;
	sEL6900_FWvers				: 		STRING(2) ;
	xEL6900_FWvers_Busy			: 		BOOL ;
	xEL6900_FWvers_Err			: 		BOOL ;
	udiEL6900_FWvers_ErrID		: 		UDINT ;

	//Read the Number Of Connections Configured In The EL6900 Logic Terminal
	fbEL6900_StatConn_EcCoESdoRead: 	FB_EcCoESdoRead ;
	bEL6900_NoOfConnections		: 		BYTE ;
	xEL6900_NoOfConnections_Busy: 		BOOL ;
	xEL6900_NoOfConnections_Err	: 		BOOL ;
	udiEL6900_NoOfConnections_ErrID: 	UDINT ;

	//Read the Number Of Safety Groups Configured In The EL6900 Logic Terminal
	fbEL6900_SafetyGrps_EcCoESdoRead: 	FB_EcCoESdoRead ;
	bEL6900_NoOfSafetyGrps		: 		BYTE ;
	xEL6900_NoOfSafetyGrps_Busy	: 		BOOL ;
	xEL6900_NoOfSafetyGrps_Err	: 		BOOL ;
	udiEL6900_NoOfSafetyGrps_ErrID: 	UDINT ;

	//Read the Number Of Safety Function Blocks Configured In The EL6900 Logic Terminal
	fbEL6900_SafetyFBs_EcCoESdoRead: 	FB_EcCoESdoRead ;
	bEL6900_NoOfSafetyFBs		: 		BYTE ;
	xEL6900_NoOfSafetyFBs_Busy	: 		BOOL ;
	xEL6900_NoOfSafetyFBs_Err	: 		BOOL ;
	udiEL6900_NoOfSafetyFBs_ErrID: 		UDINT ;
	
	//Read the Primary Micro Controller (MC1) Temperature in DegC out of the EL6900
	fbEL6900PriMCTemp_ADSRead	: 		ADSREAD ;
	wEL6900_PriMCTemp			: 		WORD ;
	xEL6900PriMCTemp_busy		: 		BOOL ;
	xEL6900PriMCTemp_Err		: 		BOOL ;
	udiEL6900PriMCTemp_ErrID	: 		UDINT ;

	//Read the Secondary Micro Controller (MC2) Temperature in DegC out of the EL6900
	fbEL6900SecMCTemp_ADSRead	: 		ADSREAD ;
	wEL6900_SecMCTemp			: 		WORD ;
	xEL6900SecMCTemp_busy		: 		BOOL ;
	xEL6900SecMCTemp_Err		: 		BOOL ;
	udiEL6900SecMCTemp_ErrID	: 		UDINT ;

	//Read the Primary Micro Controller (MC1) Voltage in mV out of the EL6900
	fbEL6900PriMCmV_ADSRead		: 		ADSREAD ;
	wEL6900_PriMCmV				: 		WORD ;
	xEL6900PriMCmV_busy			: 		BOOL ;
	xEL6900PriMCmV_Err			: 		BOOL ;
	udiEL6900PriMCmV_ErrID		: 		UDINT ;

	//Read the Secondary Micro Controller (MC2) Voltage in mV out of the EL6900
	fbEL6900SecMCmV_ADSRead		: 		ADSREAD ;
	wEL6900_SecMCmV				: 		WORD ;
	xEL6900SecMCmV_busy			: 		BOOL ;
	xEL6900SecMCmV_Err			: 		BOOL ;
	udiEL6900SecMCmV_ErrID		: 		UDINT ;

	// EL6900: Temperature and Voltage Errors
	//There are two temperature sensors inside each Microcontroller
	fbEL6900_Error_ADSRead		: 		ADSREAD ;
	wEL6900_Error				: 		WORD ;
	xEL6900Error_busy			: 		BOOL ;
	xEL6900Error_Err			: 		BOOL ;
	udiEL6900Error_ErrID		: 		UDINT ;
END_VAR
VAR_INPUT
END_VAR

//		8-2-2012
// 		This Program has been supplied by Beckhoff Automation As-Is and is intended only as an example 
//		implementation. Functionality is not guaranteed. 
//
//IF g_bHMI_ScreenBeingDisplayed = 40 THEN
// Interval timer for CoE Reads
T1(
						IN				:= 		NOT xExecute, 
						PT				:=		T#500MS, 
						Q				=>		xExecute, 
						ET				=>		tTime1 ) ;

C1(
						CU				:= 		xExecute, 
						RESET			:= 		xReset, 
						PV				:= 		wPreset, 
						Q				=> 		xDone, 
						CV				=> 		wCount) ;

IF C1.CV > 6 	THEN xReset := 1 ;
				ELSE xReset := 0 ; 
END_IF ;

// Read the serial number out of the EL6900
fbEL6900Sn_ADSRead(
						NETID			:= 		gc_sADSNetID, 
						PORT			:= 		gc_uiEL6900_EtherCATAdr, 
						IDXGRP			:= 		16#F302, 
						IDXOFFS			:= 		16#F9800002, 
						LEN				:= 		4, 
						DESTADDR		:= 		ADR(dwEL6900_Sn), 
						READ			:= 		xExecute, 
						TMOUT			:= 		T#2S, 
						BUSY			=> 		xEL6900Sn_busy, 
						ERR				=> 		xEL6900Sn_Err, 
						ERRID			=> 		xEL6900Sn_ErrID );

g_dwHMI_EL6900Sn 						:= 		dwEL6900_Sn ;

// Read the DIP Switch Setting out of the EL6900
IF C1.CV = 1 THEN
fbEL6900DSw_ADSRead(
						NETID			:= 		gc_sADSNetID, 
						PORT			:= 		gc_uiEL6900_EtherCATAdr, 
						IDXGRP			:= 		16#F302, 
						IDXOFFS			:= 		16#F9800001, 
						LEN				:= 		2, 
						DESTADDR		:= 		ADR(wEL6900_DSw), 
						READ			:= 		xExecute, 
						TMOUT			:= 		T#2S, 
						BUSY			=> 		xEL6900DSw_busy, 
						ERR				=> 		xEL6900DSw_Err, 
						ERRID			=> 		udiEL6900DSw_ErrID );

g_wHMI_EL6900DSw 						:= 		wEL6900_DSw ;
END_IF ;						

//Read the Hardware Version of the EL6900 Logic Terminal
fbEL6900_HWvers_EcCoESdoRead(
						sNetId			:= 		gc_sADSNetID, 
						nSlaveAddr		:= 		gc_uiEL6900_EtherCATAdr, 
						nSubIndex		:= 		0, 
						nIndex			:= 		16#1009, 
						pDstBuf			:=  	ADR(sEL6900_HWvers),
						cbBufLen		:= 		SIZEOF(sEL6900_HWvers), 
						bExecute		:= 		xExecute, 
						tTimeout		:= 		T#2S, 
						bBusy			=> 		xEL6900_HWvers_Busy, 
						bError			=> 		xEL6900_HWvers_Err, 
						nErrId			=> 		udiEL6900_HWvers_ErrID ) ;

g_sHMI_EL6900_HWvers					:= 		sEL6900_HWvers ;

//Read the Software Version of the EL6900 Logic Terminal (It's f/w)
fbEL6900_FWvers_EcCoESdoRead(
						sNetId			:= 		gc_sADSNetID, 
						nSlaveAddr		:= 		gc_uiEL6900_EtherCATAdr, 
						nSubIndex		:= 		0, 
						nIndex			:= 		16#100A, 
						pDstBuf			:=  	ADR(sEL6900_FWvers),
						cbBufLen		:= 		SIZEOF(sEL6900_FWvers), 
						bExecute		:= 		xExecute, 
						tTimeout		:= 		T#2S, 
						bBusy			=> 		xEL6900_FWvers_Busy, 
						bError			=> 		xEL6900_FWvers_Err, 
						nErrId			=> 		udiEL6900_FWvers_ErrID ) ;

g_sHMI_EL6900_FWvers					:= 		sEL6900_FWvers ;

//Read the Number Of Connections Configured In The EL6900 Logic Terminal
fbEL6900_StatConn_EcCoESdoRead(
						sNetId			:= 		gc_sADSNetID, 
						nSlaveAddr		:= 		gc_uiEL6900_EtherCATAdr, 
						nSubIndex		:= 		0, 
						nIndex			:= 		16#2110, 
						pDstBuf			:=  	ADR(bEL6900_NoOfConnections),
						cbBufLen		:= 		SIZEOF(bEL6900_NoOfConnections), 
						bExecute		:= 		xExecute, 
						tTimeout		:= 		T#2S, 
						bBusy			=> 		xEL6900_NoOfConnections_Busy, 
						bError			=> 		xEL6900_NoOfConnections_Err, 
						nErrId			=> 		udiEL6900_NoOfConnections_ErrID ) ;

g_bHMI_EL6900_NoOfConnections			:= 		bEL6900_NoOfConnections ;					

//Read the Number Of Safety Groups Configured In The EL6900 Logic Terminal
fbEL6900_SafetyGrps_EcCoESdoRead(
						sNetId			:= 		gc_sADSNetID, 
						nSlaveAddr		:= 		gc_uiEL6900_EtherCATAdr, 
						nSubIndex		:= 		0, 
						nIndex			:= 		16#2120, 
						pDstBuf			:=  	ADR(bEL6900_NoOfSafetyGrps),
						cbBufLen		:= 		SIZEOF(bEL6900_NoOfSafetyGrps), 
						bExecute		:= 		xExecute, 
						tTimeout		:= 		T#2S, 
						bBusy			=> 		xEL6900_NoOfSafetyGrps_Busy, 
						bError			=> 		xEL6900_NoOfSafetyGrps_Err, 
						nErrId			=> 		udiEL6900_NoOfSafetyGrps_ErrID ) ;

g_bHMI_EL6900_NoOfSafetyGrps			:= 		bEL6900_NoOfSafetyGrps ;

//Read the Number Of Safety Function Blocks Configured In The EL6900 Logic Terminal
fbEL6900_SafetyFBs_EcCoESdoRead(
						sNetId			:= 		gc_sADSNetID, 
						nSlaveAddr		:= 		gc_uiEL6900_EtherCATAdr, 
						nSubIndex		:= 		0, 
						nIndex			:= 		16#2130, 
						pDstBuf			:=  	ADR(bEL6900_NoOfSafetyFBs),
						cbBufLen		:= 		SIZEOF(bEL6900_NoOfSafetyFBs), 
						bExecute		:= 		xExecute, 
						tTimeout		:= 		T#2S, 
						bBusy			=> 		xEL6900_NoOfSafetyFBs_Busy, 
						bError			=> 		xEL6900_NoOfSafetyFBs_Err, 
						nErrId			=> 		udiEL6900_NoOfSafetyFBs_ErrID ) ;

g_bHMI_EL6900_NoOfSafetyFBs			:= 		bEL6900_NoOfSafetyFBs ;

// Read the Primary Micro Controller (MC1) Temperature in DegC out of the EL6900
IF C1.CV = 2 THEN
fbEL6900PriMCTemp_ADSRead(
						NETID			:= 		gc_sADSNetID, 
						PORT			:= 		gc_uiEL6900_EtherCATAdr, 
						IDXGRP			:= 		16#F302, 
						IDXOFFS			:= 		16#FA800001, 
						LEN				:= 		2, 
						DESTADDR		:= 		ADR(wEL6900_PriMCTemp), 
						READ			:= 		xExecute, 
						TMOUT			:= 		T#2S, 
						BUSY			=> 		xEL6900PriMCTemp_busy, 
						ERR				=> 		xEL6900PriMCTemp_Err, 
						ERRID			=> 		udiEL6900PriMCTemp_ErrID );

g_wHMI_EL6900PriMCTemp 						:= 		wEL6900_PriMCTemp ;
END_IF ;

// Read the Secondary Micro Controller (MC2) Temperature in DegC out of the EL6900
IF C1.CV = 3 THEN
fbEL6900SecMCTemp_ADSRead(
						NETID			:= 		gc_sADSNetID, 
						PORT			:= 		gc_uiEL6900_EtherCATAdr, 
						IDXGRP			:= 		16#F302, 
						IDXOFFS			:= 		16#FA800002, 
						LEN				:= 		2, 
						DESTADDR		:= 		ADR(wEL6900_SecMCTemp), 
						READ			:= 		xExecute, 
						TMOUT			:= 		T#2S, 
						BUSY			=> 		xEL6900SecMCTemp_busy, 
						ERR				=> 		xEL6900SecMCTemp_Err, 
						ERRID			=> 		udiEL6900SecMCTemp_ErrID );

g_wHMI_EL6900SecMCTemp 						:= 		wEL6900_SecMCTemp ;
END_IF ;

// Read the Primary Micro Controller (MC1) Voltage in mV out of the EL6900
IF C1.CV = 4 THEN
fbEL6900PriMCmV_ADSRead(
						NETID			:= 		gc_sADSNetID, 
						PORT			:= 		gc_uiEL6900_EtherCATAdr, 
						IDXGRP			:= 		16#F302, 
						IDXOFFS			:= 		16#FA800003, 
						LEN				:= 		2, 
						DESTADDR		:= 		ADR(wEL6900_PriMCmV), 
						READ			:= 		xExecute, 
						TMOUT			:= 		T#2S, 
						BUSY			=> 		xEL6900PriMCmV_busy, 
						ERR				=> 		xEL6900PriMCmV_Err, 
						ERRID			=> 		udiEL6900PriMCmV_ErrID );

g_wHMI_EL6900PriMC_Volts				:= 		WORD_TO_LREAL(wEL6900_PriMCmV) / 1000.0 ;
END_IF ;

// Read the Secondary Micro Controller (MC2) Voltage in mV out of the EL6900
IF C1.CV = 5 THEN
fbEL6900SecMCmV_ADSRead(
						NETID			:= 		gc_sADSNetID, 
						PORT			:= 		gc_uiEL6900_EtherCATAdr, 
						IDXGRP			:= 		16#F302, 
						IDXOFFS			:= 		16#FA800004, 
						LEN				:= 		2, 
						DESTADDR		:= 		ADR(wEL6900_SecMCmV), 
						READ			:= 		xExecute, 
						TMOUT			:= 		T#2S, 
						BUSY			=> 		xEL6900SecMCmV_busy, 
						ERR				=> 		xEL6900SecMCmV_Err, 
						ERRID			=> 		udiEL6900SecMCmV_ErrID );
			
g_wHMI_EL6900SecMC_Volts 				:= 		WORD_TO_LREAL(wEL6900_SecMCmV) / 1000.0 ;
END_IF ;
//	ELSE xReset := 1 ;
//	END_IF ;

//EL6900: Temperature and Voltage Errors
//There are two temperature sensors inside each Microcontroller
fbEL6900_Error_ADSRead(
						NETID			:= 		gc_sADSNetID, 
						PORT			:= 		gc_uiEL6900_EtherCATAdr, 
						IDXGRP			:= 		16#F302, 
						IDXOFFS			:= 		16#FA000003, 
						LEN				:= 		2, 
						DESTADDR		:= 		ADR(wEL6900_Error), 
						READ			:= 		xExecute, 
						TMOUT			:= 		T#2S, 
						BUSY			=> 		xEL6900Error_busy, 
						ERR				=> 		xEL6900Error_Err, 
						ERRID			=> 		udiEL6900Error_ErrID );
			
//These errors may only be present temporarily so they need to be latched and then cleared
//to be properly noted by the operator
g_xHMI_EL6900_MaxTemp				:= 		(wEL6900_Error = 5) OR (g_xHMI_EL6900_MaxTemp AND NOT g_xHMI_EL6900_ErrClearPB) ;
g_xHMI_EL6900_MinTemp				:= 		(wEL6900_Error = 6) OR (g_xHMI_EL6900_MinTemp AND NOT g_xHMI_EL6900_ErrClearPB) ;
g_xHMI_EL6900_TempDiffExceeded		:= 		(wEL6900_Error = 7) OR (g_xHMI_EL6900_TempDiffExceeded AND NOT g_xHMI_EL6900_ErrClearPB) ;
g_xHMI_EL6900_MaxVccMC1				:= 		(wEL6900_Error = 257) OR (g_xHMI_EL6900_MaxVccMC1 AND NOT g_xHMI_EL6900_ErrClearPB) ;
g_xHMI_EL6900_MaxVccMC2				:= 		(wEL6900_Error = 258) OR (g_xHMI_EL6900_MaxVccMC2 AND NOT g_xHMI_EL6900_ErrClearPB) ;
g_xHMI_EL6900_MinVccMC1				:= 		(wEL6900_Error = 259) OR (g_xHMI_EL6900_MinVccMC1 AND NOT g_xHMI_EL6900_ErrClearPB) ;
g_xHMI_EL6900_MinVccMC2				:= 		(wEL6900_Error = 260) OR (g_xHMI_EL6900_MinVccMC2 AND NOT g_xHMI_EL6900_ErrClearPB) ;

//Sum of all errors we know of in the EL6930 terminal
IF 		g_xHMI_EL6900_MaxTemp 
	OR 	g_xHMI_EL6900_MinTemp
	OR 	g_xHMI_EL6900_TempDiffExceeded 
	OR 	g_xHMI_EL6900_MaxVccMC1
	OR 	g_xHMI_EL6900_MaxVccMC2
	OR 	g_xHMI_EL6900_MinVccMC1
	OR 	g_xHMI_EL6900_MinVccMC2
		THEN g_xHMI_EL6900_General_Error := TRUE ;
		ELSE g_xHMI_EL6900_General_Error := FALSE ;
END_IF ;

END_PROGRAM

// ---- POUs/Safety_Diagnostics/EL1904_ADS_Reads.TcPOU
PROGRAM EL1904_ADS_Reads
VAR
//		8-2-2012
// 		This Program has been supplied by Beckhoff Automation As-Is and is intended only as an example 
//		implementation. Functionality is not guaranteed. 
//
	//Time to check CoE values (Every 2 seconds in this case)
	T1							: 		TON ;
	xExecute					: 		BOOL ;
	tTime1						: 		TIME ;

	//Counter for just some very simple sequencing
	C1							: 		CTU ;
	xReset						: 		BOOL ;
	wPreset						: 		WORD := 10 ;
	xDone						: 		BOOL ;
	wCount						: 		WORD ;
	
	//Get EL1904 terminal's serial number
	fbEL1904Sn_ADSRead			: 		ADSREAD ;
	dwEL1904_Sn					: 		DWORD ;
	xEL1904Sn_busy				: 		BOOL ;
	xEL1904Sn_Err				: 		BOOL ;
	xEL1904Sn_ErrID				: 		UDINT ;

	//Get EL1904 terminal's DIP switch setting
	fbEL1904DSw_ADSRead			: 		ADSREAD ;
	wEL1904_DSw					: 		WORD ;
	xEL1904DSw_busy				: 		BOOL ;
	xEL1904DSw_Err				: 		BOOL ;
	udiEL1904DSw_ErrID			: 		UDINT ;

	//Read the Hardware Version of the EL1904 Terminal
	fbEL1904_HWvers_EcCoESdoRead: 		FB_EcCoESdoRead ;
	sEL1904_HWvers				: 		STRING(2) ;
	xEL1904_HWvers_Busy			: 		BOOL ;
	xEL1904_HWvers_Err			: 		BOOL ;
	udiEL1904_HWvers_ErrID		: 		UDINT ;

	//Read the Software Version of the EL1904 Terminal (It's f/w)
	fbEL1904_FWvers_EcCoESdoRead: 		FB_EcCoESdoRead ;
	sEL1904_FWvers				: 		STRING(2) ;
	xEL1904_FWvers_Busy			: 		BOOL ;
	xEL1904_FWvers_Err			: 		BOOL ;
	udiEL1904_FWvers_ErrID		: 		UDINT ;

	//EL1904 FEATURES: Operating Mode
	fbEL1904_OperatingMode_ADSRead	: 	ADSREAD ;
	wEL1904_OperMode				: 	WORD ;
	xEL1904_OperMode_busy			: 	BOOL ;
	xEL1904_OperMode_Err			: 	BOOL ;
	udiEL1904_OperModeID			: 	UDINT ;

	//Sequence through 0x8001 FS Sensor Test
	iFS_Sensor_Test					: 	INT ;

	//EL1904 FEATURES: Sensor Test Channel 1 Active/Inactive
	fbEL1904_STActive1_EcCoESdoRead	: 	FB_EcCoESdoRead ;
	bEL1904_STActive1				: 	BYTE ;
	xEL1904_STActive1_busy			: 	BOOL ;
	xEL1904_STActive1_Err			: 	BOOL ;
	udiEL1904_STActive1ID			: 	UDINT ;
	iCaseZeroScans					: 	INT ;
	
	// EL1904 FEATURES: Sensor Test Channel 2 Active/Inactive
	fbEL1904_STActive2_EcCoESdoRead	: 	FB_EcCoESdoRead ;
	bEL1904_STActive2				: 	BYTE ;
	xEL1904_STActive2				: 	BOOL ;
	xEL1904_STActive2_busy			: 	BOOL ;
	xEL1904_STActive2_Err			: 	BOOL ;
	udiEL1904_STActive2ID			: 	UDINT ;
	iCaseOneScans					: 	INT ;

	// EL1904 FEATURES: Sensor Test Channel 3 Active/Inactive	
	fbEL1904_STActive3_EcCoESdoRead	: 	FB_EcCoESdoRead ;
	bEL1904_STActive3				: 	BYTE ;
	xEL1904_STActive3_busy			: 	BOOL ;
	xEL1904_STActive3_Err			: 	BOOL ;
	udiEL1904_STActive3ID			: 	UDINT ;
	iCaseTwoScans					: 	INT ;

	// EL1904 FEATURES: Sensor Test Channel 4 Active/Inactive	
	fbEL1904_STActive4_EcCoESdoRead	: 	FB_EcCoESdoRead ;
	bEL1904_STActive4				: 	BYTE ;
	xEL1904_STActive4_busy			: 	BOOL ;
	xEL1904_STActive4_Err			: 	BOOL ;
	udiEL1904_STActive4ID			: 	UDINT ;
	iCaseThreeScans					: 	INT ;

	//Sequence through 0x8002 FS Logic Of Input Pairs
	iFS_LogicOfInputPairs			: 	INT ;

	// EL1904 FEATURES: Logic of Channels 1 and 2	
	fbEL1904_Logic1_2_EcCoESdoRead	: 	FB_EcCoESdoRead ;
	bEL1904_Logic1_2				: 	BYTE ;
	xEL1904_Logic1_2_busy			: 	BOOL ;
	xEL1904_Logic1_2_Err			: 	BOOL ;
	udiEL1904_Logic1_2ID			: 	UDINT ;
	iCaseLogicZeroScans				: 	INT ;

	// EL1904 FEATURES: Logic of Channels 3 and 4	
	fbEL1904_Logic3_4_EcCoESdoRead	: 	FB_EcCoESdoRead ;
	bEL1904_Logic3_4				: 	BYTE ;
	xEL1904_Logic3_4_busy			: 	BOOL ;
	xEL1904_Logic3_4_Err			: 	BOOL ;
	udiEL1904_Logic3_4ID			: 	UDINT ;
	iCaseLogicOneScans				: 	INT ;
	
	//Get EL1904 terminal's MC1 temperature (in Deg C)
	fbEL1904PriMCTemp_ADSRead	: 		ADSREAD ;
	wEL1904_PriMCTemp			: 		WORD ;
	xEL1904PriMCTemp_busy		: 		BOOL ;
	xEL1904PriMCTemp_Err		: 		BOOL ;
	udiEL1904PriMCTemp_ErrID	: 		UDINT ;
	
	//Get EL1904 terminal's MC2 termperature (in Deg C)
	fbEL1904SecMCTemp_ADSRead	: 		ADSREAD ;
	wEL1904_SecMCTemp			: 		WORD ;
	xEL1904SecMCTemp_busy		: 		BOOL ;
	xEL1904SecMCTemp_Err		: 		BOOL ;
	udiEL1904SecMCTemp_ErrID	: 		UDINT ;

	//Get EL1904 terminal's MC1 voltage (in mV)
	fbEL1904PriMCmV_ADSRead		: 		ADSREAD ;
	wEL1904_PriMCmV				: 		WORD ;
	xEL1904PriMCmV_busy			: 		BOOL ;
	xEL1904PriMCmV_Err			: 		BOOL ;
	udiEL1904PriMCmV_ErrID		: 		UDINT ;
	q_wHMI_EL1904PriMCmV		: 		LREAL ;

	//Get EL1904 terminal's MC2 voltage (in mV)
	fbEL1904SecMCmV_ADSRead		: 		ADSREAD ;
	wEL1904_SecMCmV				: 		WORD ;
	xEL1904SecMCmV_busy			: 		BOOL ;
	xEL1904SecMCmV_Err			: 		BOOL ;
	udiEL1904SecMCmV_ErrID		: 		UDINT ;
	//
	// EL1904 ALARMS
	//
		//Get EL1904 Diagnostic object 800E:0A - Sensor Test Errors
	fbEL1904SensT_ADSRead		: 		ADSREAD ;
	wEL1904SenT					: 		WORD ;
	wEL1904_SenT				: 		WORD ;
	xEL1904SenT_busy			: 		BOOL ;
	xEL1904SenT_Err				: 		BOOL ;
	udiEL1904SenT_ErrID			: 		UDINT ;

	//Get EL1904 Diagnostic object 800E:0B - Error During Two-Channel Evaluation
	fbEL1904_2CHEval_ADSRead	: 		ADSREAD ;
	wEL1904_2CHEval				: 		WORD ;
	xEL1904_2CHEval_busy		: 		BOOL ;
	xEL1904_2CHEval_Err			: 		BOOL ;
	udiEL1904_2CHEval_ErrID		: 		UDINT ;

	//Get EL1904 Diagnostic object 800E:0C - Error In Safety Mat Operating Mode: Input Pair Disagree
	fbEL1904_SMiPair_ADSRead	: 		ADSREAD ;
	wEL1904_SMiPair				: 		WORD ;
	xEL1904_SMiPair_busy		: 		BOOL ;
	xEL1904_SMiPair_Err			: 		BOOL ;
	udiEL1904_SMiPair_ErrID		: 		UDINT ;

	//Get EL1904 Diagnostic object 800E:0D - Error In Safety Mat Operating Mode: External Supply (No test pulses)
	fbEL1904_SMExtSupply_ADSRead: 		ADSREAD ;
	wEL1904_SMExtSupply			: 		WORD ;
	xEL1904_SMExtSupply_busy	: 		BOOL ;
	xEL1904_SMExtSupply_Err		: 		BOOL ;
	udiEL1904_SMExtSupply_ErrID	: 		UDINT ;
END_VAR

//		8-2-2012
// 		This Program has been supplied by Beckhoff Automation As-Is and is intended only as an example 
//		implementation. Functionality is not guaranteed. 
//
//IF g_bHMI_ScreenBeingDisplayed = 10 THEN
// Interval timer for CoE Reads
T1(
						IN				:= 		NOT xExecute, 
						PT				:=		T#500MS, 
						Q				=>		xExecute, 
						ET				=>		tTime1 ) ;

C1(
						CU				:= 		xExecute, 
						RESET			:= 		xReset, 
						PV				:= 		wPreset, 
						Q				=> 		xDone, 
						CV				=> 		wCount) ;

IF C1.CV > 6 	THEN xReset := 1 ;
				ELSE xReset := 0 ; 
END_IF ;
						
// Read the serial number out of the EL1904
fbEL1904Sn_ADSRead(
						NETID			:= 		gc_sADSNetID, 
						PORT			:= 		gc_uiEL1904_EtherCATAdr, 
						IDXGRP			:= 		16#F302, 
						IDXOFFS			:= 		16#F9800002, 
						LEN				:= 		4, 
						DESTADDR		:= 		ADR(dwEL1904_Sn), 
						READ			:= 		xExecute, 
						TMOUT			:= 		T#2S, 
						BUSY			=> 		xEL1904Sn_busy, 
						ERR				=> 		xEL1904Sn_Err, 
						ERRID			=> 		xEL1904Sn_ErrID );

g_dwHMI_EL1904Sn 						:= 		dwEL1904_Sn ;

// Read the DIP Switch Setting out of the EL1904
IF C1.CV = 1 THEN
fbEL1904DSw_ADSRead(
						NETID			:= 		gc_sADSNetID, 
						PORT			:= 		gc_uiEL1904_EtherCATAdr, 
						IDXGRP			:= 		16#F302, 
						IDXOFFS			:= 		16#F9800001, 
						LEN				:= 		2, 
						DESTADDR		:= 		ADR(wEL1904_DSw), 
						READ			:= 		xExecute, 
						TMOUT			:= 		T#2S, 
						BUSY			=> 		xEL1904DSw_busy, 
						ERR				=> 		xEL1904DSw_Err, 
						ERRID			=> 		udiEL1904DSw_ErrID );

g_wHMI_EL1904DSw 						:= 		wEL1904_DSw ;
END_IF ;

//Read the Hardware Version of the EL1904 Terminal
fbEL1904_HWvers_EcCoESdoRead(
						sNetId			:= 		gc_sADSNetID, 
						nSlaveAddr		:= 		gc_uiEL1904_EtherCATAdr, 
						nSubIndex		:= 		0, 
						nIndex			:= 		16#1009, 
						pDstBuf			:=  	ADR(sEL1904_HWvers),
						cbBufLen		:= 		SIZEOF(sEL1904_HWvers), 
						bExecute		:= 		xExecute, 
						tTimeout		:= 		T#2S, 
						bBusy			=> 		xEL1904_HWvers_Busy, 
						bError			=> 		xEL1904_HWvers_Err, 
						nErrId			=> 		udiEL1904_HWvers_ErrID ) ;

g_sHMI_EL1904_HWvers					:= 		sEL1904_HWvers ;

//Read the Software Version of the EL1904 Logic Terminal (It's f/w)
fbEL1904_FWvers_EcCoESdoRead(
						sNetId			:= 		gc_sADSNetID, 
						nSlaveAddr		:= 		gc_uiEL1904_EtherCATAdr, 
						nSubIndex		:= 		0, 
						nIndex			:= 		16#100A, 
						pDstBuf			:=  	ADR(sEL1904_FWvers),
						cbBufLen		:= 		SIZEOF(sEL1904_FWvers), 
						bExecute		:= 		xExecute, 
						tTimeout		:= 		T#2S, 
						bBusy			=> 		xEL1904_FWvers_Busy, 
						bError			=> 		xEL1904_FWvers_Err, 
						nErrId			=> 		udiEL1904_FWvers_ErrID ) ;

g_sHMI_EL1904_FWvers					:= 		sEL1904_FWvers ;

// EL1904 FEATURES: Operating Mode
fbEL1904_OperatingMode_ADSRead(
						NETID			:= 		gc_sADSNetID, 
						PORT			:= 		gc_uiEL1904_EtherCATAdr, 
						IDXGRP			:= 		16#F302, 
						IDXOFFS			:= 		16#80000001, 
						LEN				:= 		2, 
						DESTADDR		:=		ADR(wEL1904_OperMode), 
						READ			:= 		xExecute, 
						TMOUT			:= 		T#2S, 
						BUSY			=> 		xEL1904_OperMode_busy, 
						ERR				=> 		xEL1904_OperMode_Err, 
						ERRID			=> 		udiEL1904_OperModeID );
		
IF wEL1904_OperMode 					= 		0 THEN
	g_sHMI_EL1904_OperatingMode 		:= 		'Digital' ;
	ELSIF wEL1904_OperMode 				= 		1 THEN
	g_sHMI_EL1904_OperatingMode 		:= 		'Standstill Monitoring 1' ;
	ELSIF wEL1904_OperMode 				= 		2 THEN
	g_sHMI_EL1904_OperatingMode 		:= 		'Standstill Monitoring 2' ;
ELSE
	g_sHMI_EL1904_OperatingMode 		:= 		'Invalid Mode' ;
END_IF ;

CASE iFS_Sensor_Test OF

0:
// EL1904 FEATURES: Sensor Test Channel 1 Active/Inactive
iCaseThreeScans 						:= 		0 ;
fbEL1904_STActive1_EcCoESdoRead(
						sNetId			:= 		gc_sADSNetID, 
						nSlaveAddr		:= 		gc_uiEL1904_EtherCATAdr, 
						nSubIndex		:= 		1, 
						nIndex			:= 		16#8001, 
						pDstBuf			:= 		ADR(bEL1904_STActive1), 
						cbBufLen		:= 		SIZEOF(bEL1904_STActive1), 
						bExecute		:= 		xExecute, 
						tTimeout		:= 		T#2S, 
						bBusy			=> 		xEL1904_STActive1_busy, 
						bError			=> 		xEL1904_STActive1_Err, 
						nErrId			=> 		udiEL1904_STActive1ID );

g_xHMI_EL1904_SensTestActive1			:= 		bEL1904_STActive1.0 ;

iCaseZeroScans := iCaseZeroScans + 1 ; //Prevent code from passing through in only one pass

IF NOT xEL1904_STActive1_busy AND NOT xEL1904_STActive1_Err AND iCaseZeroScans <> 0 THEN
	iFS_Sensor_Test := 1 ;
END_IF ;

1:
// EL1904 FEATURES: Sensor Test Channel 2 Active/Inactive
iCaseZeroScans 							:= 		0 ;
fbEL1904_STActive2_EcCoESdoRead(
						sNetId			:= 		gc_sADSNetID, 
						nSlaveAddr		:= 		gc_uiEL1904_EtherCATAdr, 
						nSubIndex		:= 		2, 
						nIndex			:= 		16#8001, 
						pDstBuf			:= 		ADR(bEL1904_STActive2), 
						cbBufLen		:= 		SIZEOF(bEL1904_STActive2), 
						bExecute		:= 		xExecute, 
						tTimeout		:= 		T#2S, 
						bBusy			=> 		xEL1904_STActive2_busy, 
						bError			=> 		xEL1904_STActive2_Err, 
						nErrId			=> 		udiEL1904_STActive2ID );

g_xHMI_EL1904_SensTestActive2			:= 		bEL1904_STActive2.0 ;

iCaseOneScans := iCaseOneScans + 1 ; //Prevent code from passing through in only one pass

IF NOT xEL1904_STActive2_busy AND NOT xEL1904_STActive2_Err AND iCaseOneScans <> 0 THEN
	iFS_Sensor_Test := 2 ;
END_IF ;

2:
// EL1904 FEATURES: Sensor Test Channel 3 Active/Inactive
iCaseOneScans 							:= 		0 ;
fbEL1904_STActive3_EcCoESdoRead(
						sNetId			:= 		gc_sADSNetID, 
						nSlaveAddr		:= 		gc_uiEL1904_EtherCATAdr, 
						nSubIndex		:= 		3, 
						nIndex			:= 		16#8001, 
						pDstBuf			:= 		ADR(bEL1904_STActive3), 
						cbBufLen		:= 		SIZEOF(bEL1904_STActive3), 
						bExecute		:= 		xExecute, 
						tTimeout		:= 		T#2S, 
						bBusy			=> 		xEL1904_STActive3_busy, 
						bError			=> 		xEL1904_STActive3_Err, 
						nErrId			=> 		udiEL1904_STActive3ID );

g_xHMI_EL1904_SensTestActive3			:= 		bEL1904_STActive3.0 ;

iCaseTwoScans := iCaseTwoScans + 1 ; //Prevent code from passing through in only one pass

IF NOT xEL1904_STActive3_busy AND NOT xEL1904_STActive3_Err AND iCaseTwoScans <> 0 THEN
	iFS_Sensor_Test := 3 ;
END_IF ;

3:
// EL1904 FEATURES: Sensor Test Channel 4 Active/Inactive
iCaseTwoScans 							:= 		0 ;
fbEL1904_STActive4_EcCoESdoRead(
						sNetId			:= 		gc_sADSNetID, 
						nSlaveAddr		:= 		gc_uiEL1904_EtherCATAdr, 
						nSubIndex		:= 		4, 
						nIndex			:= 		16#8001, 
						pDstBuf			:= 		ADR(bEL1904_STActive4), 
						cbBufLen		:= 		SIZEOF(bEL1904_STActive4), 
						bExecute		:= 		xExecute, 
						tTimeout		:= 		T#2S, 
						bBusy			=> 		xEL1904_STActive4_busy, 
						bError			=> 		xEL1904_STActive4_Err, 
						nErrId			=> 		udiEL1904_STActive4ID );

g_xHMI_EL1904_SensTestActive4			:= 		bEL1904_STActive4.0 ;

iCaseThreeScans := iCaseThreeScans + 1 ; //Prevent code from passing through in only one pass

IF NOT xEL1904_STActive4_busy AND NOT xEL1904_STActive4_Err AND iCaseThreeScans <> 0 THEN
	iFS_Sensor_Test := 0 ;
END_IF ;
	END_CASE ;

//Sequence through 0x8002 FS Logic Of Input Pairs
CASE iFS_LogicOfInputPairs OF

0:
// EL1904 FEATURES: Logic of Channels 1 and 2
iCaseLogicOneScans 						:= 		0 ;
fbEL1904_Logic1_2_EcCoESdoRead(
						sNetId			:= 		gc_sADSNetID, 
						nSlaveAddr		:= 		gc_uiEL1904_EtherCATAdr, 
						nSubIndex		:= 		1, 
						nIndex			:= 		16#8002, 
						pDstBuf			:= 		ADR(bEL1904_Logic1_2), 
						cbBufLen		:= 		SIZEOF(bEL1904_Logic1_2), 
						bExecute		:= 		xExecute, 
						tTimeout		:= 		T#2S, 
						bBusy			=> 		xEL1904_Logic1_2_busy, 
						bError			=> 		xEL1904_Logic1_2_Err, 
						nErrId			=> 		udiEL1904_Logic1_2ID );

IF bEL1904_Logic1_2 					= 		0 THEN
	g_sHMI_EL1904_LogicCh1andCh2 		:= 		'Single Channel Logic' ;
	ELSIF bEL1904_Logic1_2 				= 		1 THEN
	g_sHMI_EL1904_LogicCh1andCh2 		:= 		'Asynchronous Repetitive OSSD, Sensor Test Must Be Disabled!' ;
	ELSIF bEL1904_Logic1_2 				= 		2 THEN
	g_sHMI_EL1904_LogicCh1andCh2 		:= 		'Any Pulse Repetitive OSSD, Sensor Test Must Be Disabled!' ;
	ELSIF bEL1904_Logic1_2 				= 		3 THEN
	g_sHMI_EL1904_LogicCh1andCh2 		:= 		'Short Cut, No Module Fault' ;
ELSE
	g_sHMI_EL1904_LogicCh1andCh2 		:= 		'Invalid Logic CH1 and CH2' ;
END_IF ;						

iCaseLogicZeroScans := iCaseLogicZeroScans + 1 ; //Prevent code from passing through in only one pass

IF NOT xEL1904_Logic1_2_busy AND NOT xEL1904_Logic1_2_Err AND iCaseLogicZeroScans <> 0 THEN
	iFS_LogicOfInputPairs := 1 ;
END_IF ;

1:						
// EL1904 FEATURES: Logic of Channels 3 and 4
iCaseLogicZeroScans 					:= 		0 ;
fbEL1904_Logic3_4_EcCoESdoRead(
						sNetId			:= 		gc_sADSNetID, 
						nSlaveAddr		:= 		gc_uiEL1904_EtherCATAdr, 
						nSubIndex		:= 		3, 
						nIndex			:= 		16#8002, 
						pDstBuf			:= 		ADR(bEL1904_Logic3_4), 
						cbBufLen		:= 		SIZEOF(bEL1904_Logic3_4), 
						bExecute		:= 		xExecute, 
						tTimeout		:= 		T#2S, 
						bBusy			=> 		xEL1904_Logic3_4_busy, 
						bError			=> 		xEL1904_Logic3_4_Err, 
						nErrId			=> 		udiEL1904_Logic3_4ID );

IF bEL1904_Logic3_4 					= 		0 THEN
	g_sHMI_EL1904_LogicCh3andCh4 		:= 		'Single Channel Logic' ;
	ELSIF bEL1904_Logic3_4  			= 		1 THEN
	g_sHMI_EL1904_LogicCh3andCh4 		:= 		'Asynchronous Repetitive OSSD, Sensor Test Must Be Disabled!' ;
	ELSIF bEL1904_Logic3_4 				= 		2 THEN
	g_sHMI_EL1904_LogicCh3andCh4 		:= 		'Any Pulse Repetitive OSSD, Sensor Test Must Be Disabled!' ;
	ELSIF bEL1904_Logic3_4  			= 		3 THEN
	g_sHMI_EL1904_LogicCh3andCh4 		:= 		'Short Cut, No Module Fault' ;
ELSE
	g_sHMI_EL1904_LogicCh3andCh4 		:= 		'Invalid Logic CH3 and CH4' ;
	END_IF ;						

iCaseLogicOneScans := iCaseLogicOneScans + 1 ; //Prevent code from passing through in only one pass

IF NOT xEL1904_Logic3_4_busy AND NOT xEL1904_Logic3_4_Err AND iCaseLogicOneScans <> 0 THEN
	iFS_LogicOfInputPairs := 0 ;
END_IF ;
	END_CASE ;

// Read the Primary Micro Controller (MC1) Temperature in DegC out of the EL1904
IF C1.CV = 2 THEN
fbEL1904PriMCTemp_ADSRead(
						NETID			:= 		gc_sADSNetID, 
						PORT			:= 		gc_uiEL1904_EtherCATAdr, 
						IDXGRP			:= 		16#F302, 
						IDXOFFS			:= 		16#FA800001, 
						LEN				:= 		2, 
						DESTADDR		:= 		ADR(wEL1904_PriMCTemp), 
						READ			:= 		xExecute, 
						TMOUT			:= 		T#2S, 
						BUSY			=> 		xEL1904PriMCTemp_busy, 
						ERR				=> 		xEL1904PriMCTemp_Err, 
						ERRID			=> 		udiEL1904PriMCTemp_ErrID );

g_wHMI_EL1904PriMCTemp 						:= 		wEL1904_PriMCTemp ;
END_IF ;

// Read the Secondary Micro Controller (MC2) Temperature in DegC out of the EL1904
IF C1.CV = 3 THEN
fbEL1904SecMCTemp_ADSRead(
						NETID			:= 		gc_sADSNetID, 
						PORT			:= 		gc_uiEL1904_EtherCATAdr, 
						IDXGRP			:= 		16#F302, 
						IDXOFFS			:= 		16#FA800002, 
						LEN				:= 		2, 
						DESTADDR		:= 		ADR(wEL1904_SecMCTemp), 
						READ			:= 		xExecute, 
						TMOUT			:= 		T#2S, 
						BUSY			=> 		xEL1904SecMCTemp_busy, 
						ERR				=> 		xEL1904SecMCTemp_Err, 
						ERRID			=> 		udiEL1904SecMCTemp_ErrID );

g_wHMI_EL1904SecMCTemp 						:= 		wEL1904_SecMCTemp ;
END_IF ;

// Read the Primary Micro Controller (MC1) Voltage in mV out of the EL1904
IF C1.CV = 4 THEN
fbEL1904PriMCmV_ADSRead(
						NETID			:= 		gc_sADSNetID, 
						PORT			:= 		gc_uiEL1904_EtherCATAdr, 
						IDXGRP			:= 		16#F302, 
						IDXOFFS			:= 		16#FA810001, 
						LEN				:= 		2, 
						DESTADDR		:= 		ADR(wEL1904_PriMCmV), 
						READ			:= 		xExecute, 
						TMOUT			:= 		T#2S, 
						BUSY			=> 		xEL1904PriMCmV_busy, 
						ERR				=> 		xEL1904PriMCmV_Err, 
						ERRID			=> 		udiEL1904PriMCmV_ErrID );

						
g_wHMI_EL1904PriMC_Volts				:= 		WORD_TO_LREAL(wEL1904_PriMCmV) / 1000.0 ;
END_IF ;

// Read the Secondary Micro Controller (MC2) Voltage in mV out of the EL1904
IF C1.CV = 5 THEN
fbEL1904SecMCmV_ADSRead(
						NETID			:= 		gc_sADSNetID, 
						PORT			:= 		gc_uiEL1904_EtherCATAdr, 
						IDXGRP			:= 		16#F302, 
						IDXOFFS			:= 		16#FA810002, 
						LEN				:= 		2, 
						DESTADDR		:= 		ADR(wEL1904_SecMCmV), 
						READ			:= 		xExecute, 
						TMOUT			:= 		T#2S, 
						BUSY			=> 		xEL1904SecMCmV_busy, 
						ERR				=> 		xEL1904SecMCmV_Err, 
						ERRID			=> 		udiEL1904SecMCmV_ErrID );
			
g_wHMI_EL1904SecMC_Volts 				:= 		WORD_TO_LREAL(wEL1904_SecMCmV) / 1000.0 ;
	END_IF ;
//		ELSE xReset := 1 ;
//		END_IF ;

//		
//		EL1904 ALARMS	
//	
// EL1904: Sensor Test Error
fbEL1904SensT_ADSRead(
						NETID			:= 		gc_sADSNetID, 
						PORT			:= 		gc_uiEL1904_EtherCATAdr, 
						IDXGRP			:= 		16#F302, 
						IDXOFFS			:= 		16#800E000A, 
						LEN				:= 		2, 
						DESTADDR		:= 		ADR(wEL1904_SenT), 
						READ			:= 		xExecute, 
						TMOUT			:= 		T#2S, 
						BUSY			=> 		xEL1904SenT_busy, 
						ERR				=> 		xEL1904SenT_Err, 
						ERRID			=> 		udiEL1904SenT_ErrID );

//These errors may only be present temporarily so they need to be latched and then cleared
//to be properly noted by the operator
g_xHMI_EL1904SenT1 						:= 		wEL1904_SenT.0 OR (g_xHMI_EL1904SenT1 AND NOT g_xHMI_EL1904_ErrClearPB) ;
g_xHMI_EL1904SenT2 						:= 		wEL1904_SenT.1 OR (g_xHMI_EL1904SenT2 AND NOT g_xHMI_EL1904_ErrClearPB) ;
g_xHMI_EL1904SenT3 						:= 		wEL1904_SenT.2 OR (g_xHMI_EL1904SenT3 AND NOT g_xHMI_EL1904_ErrClearPB) ;
g_xHMI_EL1904SenT4 						:= 		wEL1904_SenT.3 OR (g_xHMI_EL1904SenT4 AND NOT g_xHMI_EL1904_ErrClearPB) ;


// EL1904: 2-Channel Evaluation Error
// The two channels contradict each other (not same value)
fbEL1904_2CHEval_ADSRead(
						NETID			:= 		gc_sADSNetID, 
						PORT			:= 		gc_uiEL1904_EtherCATAdr, 
						IDXGRP			:= 		16#F302, 
						IDXOFFS			:= 		16#800E000B, 
						LEN				:= 		2, 
						DESTADDR		:= 		ADR(wEL1904_2CHEval), 
						READ			:= 		xExecute, 
						TMOUT			:= 		T#2S, 
						BUSY			=> 		xEL1904_2CHEval_busy, 
						ERR				=> 		xEL1904_2CHEval_Err, 
						ERRID			=> 		udiEL1904_2CHEval_ErrID );

//These errors may only be present temporarily so they need to be latched and then cleared
//to be properly noted by the operator
g_xHMI_EL1904_2CHEval_Pair1				:= 		wEL1904_2CHEval.0 OR (g_xHMI_EL1904_2CHEval_Pair1 AND NOT g_xHMI_EL1904_ErrClearPB) ;
g_xHMI_EL1904_2CHEval_Pair2				:= 		wEL1904_2CHEval.1 OR (g_xHMI_EL1904_2CHEval_Pair2 AND NOT g_xHMI_EL1904_ErrClearPB) ;


// EL1904: Error In Safety Mat Operating Mode
// Input pairs not in the same state (not same value)
fbEL1904_SMiPair_ADSRead(
						NETID			:= 		gc_sADSNetID, 
						PORT			:= 		gc_uiEL1904_EtherCATAdr, 
						IDXGRP			:= 		16#F302, 
						IDXOFFS			:= 		16#800E000C, 
						LEN				:= 		2, 
						DESTADDR		:= 		ADR(wEL1904_SMiPair), 
						READ			:= 		xExecute, 
						TMOUT			:= 		T#2S, 
						BUSY			=> 		xEL1904_SMiPair_busy, 
						ERR				=> 		xEL1904_SMiPair_Err, 
						ERRID			=> 		udiEL1904_SMiPair_ErrID );

//These errors may only be present temporarily so they need to be latched and then cleared
//to be properly noted by the operator
g_xHMI_EL1904_SMiPair_Pair1				:= 		(wEL1904_SMiPair.0 AND wEL1904_SMiPair.1) OR (g_xHMI_EL1904_SMiPair_Pair1 AND NOT g_xHMI_EL1904_ErrClearPB) ;
g_xHMI_EL1904_SMiPair_Pair2				:= 		(wEL1904_SMiPair.2 AND wEL1904_SMiPair.3) OR (g_xHMI_EL1904_SMiPair_Pair2 AND NOT g_xHMI_EL1904_ErrClearPB) ;


// EL1904: Error in Safety Mat Operating Supply
// External supply detected (Input channel not getting test pulses)
fbEL1904_SMExtSupply_ADSRead(
						NETID			:= 		gc_sADSNetID, 
						PORT			:= 		gc_uiEL1904_EtherCATAdr, 
						IDXGRP			:= 		16#F302, 
						IDXOFFS			:= 		16#800E000D, 
						LEN				:= 		2, 
						DESTADDR		:= 		ADR(wEL1904_SMExtSupply), 
						READ			:= 		xExecute, 
						TMOUT			:= 		T#2S, 
						BUSY			=> 		xEL1904_SMExtSupply_busy, 
						ERR				=> 		xEL1904_SMExtSupply_Err, 
						ERRID			=> 		udiEL1904_SMExtSupply_ErrID );

//These errors may only be present temporarily so they need to be latched and then cleared
//to be properly noted by the operator
g_xHMI_EL1904_SMExtSupply_CH1			:= 		wEL1904_SMExtSupply.0 OR (g_xHMI_EL1904_SMExtSupply_CH1 AND NOT g_xHMI_EL1904_ErrClearPB) ;
g_xHMI_EL1904_SMExtSupply_CH2			:= 		wEL1904_SMExtSupply.2 OR (g_xHMI_EL1904_SMExtSupply_CH2 AND NOT g_xHMI_EL1904_ErrClearPB) ;
g_xHMI_EL1904_SMExtSupply_CH3			:= 		wEL1904_SMExtSupply.3 OR (g_xHMI_EL1904_SMExtSupply_CH3 AND NOT g_xHMI_EL1904_ErrClearPB) ;
g_xHMI_EL1904_SMExtSupply_CH4			:= 		wEL1904_SMExtSupply.4 OR (g_xHMI_EL1904_SMExtSupply_CH4 AND NOT g_xHMI_EL1904_ErrClearPB) ;


//Sum of all errors we know of in the EL1904 terminal
IF 		g_xHMI_EL1904SenT1 
	OR 	g_xHMI_EL1904SenT2 
	OR 	g_xHMI_EL1904SenT3 
	OR 	g_xHMI_EL1904SenT4
	OR 	g_xHMI_EL1904_2CHEval_Pair1
	OR 	g_xHMI_EL1904_2CHEval_Pair2
	OR 	g_xHMI_EL1904_SMiPair_Pair1
	OR 	g_xHMI_EL1904_SMiPair_Pair2
	OR 	g_xHMI_EL1904_SMExtSupply_CH1
	OR 	g_xHMI_EL1904_SMExtSupply_CH2
	OR 	g_xHMI_EL1904_SMExtSupply_CH3
	OR 	g_xHMI_EL1904_SMExtSupply_CH4
		THEN g_xHMI_EL1904_General_Error := TRUE ;
		ELSE g_xHMI_EL1904_General_Error := FALSE ;
	END_IF ;

END_PROGRAM

// ---- POUs/Safety_Diagnostics/EL2904_ADS_Reads.TcPOU
PROGRAM EL2904_ADS_Reads
//		8-2-2012
// 		This Program has been supplied by Beckhoff Automation As-Is and is intended only as an example 
//		implementation. Functionality is not guaranteed. 
//
VAR
	//Time to check CoE values (Every 2 seconds in this case)
	T1							: 		TON ;
	xExecute					: 		BOOL ;
	tTime1						: 		TIME ;

	//Counter for just some very simple sequencing
	C1							: 		CTU ;
	xReset						: 		BOOL ;
	wPreset						: 		WORD := 10 ;
	xDone						: 		BOOL ;
	wCount						: 		WORD ;
	
	//Get EL2904 terminal's serial number
	fbEL2904Sn_ADSRead			: 		ADSREAD ;
	dwEL2904_Sn					: 		DWORD ;
	xEL2904Sn_busy				: 		BOOL ;
	xEL2904Sn_Err				: 		BOOL ;
	xEL2904Sn_ErrID				: 		UDINT ;

	//Get EL2904 terminal's DIP switch setting
	fbEL2904DSw_ADSRead			: 		ADSREAD ;
	wEL2904_DSw					: 		WORD ;
	xEL2904DSw_busy				: 		BOOL ;
	xEL2904DSw_Err				: 		BOOL ;
	udiEL2904DSw_ErrID			: 		UDINT ;

	//Read the Hardware Version of the EL2904 Terminal
	fbEL2904_HWvers_EcCoESdoRead: 		FB_EcCoESdoRead ;
	sEL2904_HWvers				: 		STRING(2) ;
	xEL2904_HWvers_Busy			: 		BOOL ;
	xEL2904_HWvers_Err			: 		BOOL ;
	udiEL2904_HWvers_ErrID		: 		UDINT ;

	//Read the Software Version of the EL2904 Terminal (It's f/w)
	fbEL2904_FWvers_EcCoESdoRead: 		FB_EcCoESdoRead ;
	sEL2904_FWvers				: 		STRING(2) ;
	xEL2904_FWvers_Busy			: 		BOOL ;
	xEL2904_FWvers_Err			: 		BOOL ;
	udiEL2904_FWvers_ErrID		: 		UDINT ;
	
	//Get EL1904 terminal's MC1 temperature (in Deg C)
	fbEL2904PriMCTemp_ADSRead	: 		ADSREAD ;
	wEL2904_PriMCTemp			: 		WORD ;
	xEL2904PriMCTemp_busy		: 		BOOL ;
	xEL2904PriMCTemp_Err		: 		BOOL ;
	udiEL2904PriMCTemp_ErrID	: 		UDINT ;
	
	//Get EL1904 terminal's MC2 termperature (in Deg C)
	fbEL2904SecMCTemp_ADSRead	: 		ADSREAD ;
	wEL2904_SecMCTemp			: 		WORD ;
	xEL2904SecMCTemp_busy		: 		BOOL ;
	xEL2904SecMCTemp_Err		: 		BOOL ;
	udiEL2904SecMCTemp_ErrID	: 		UDINT ;
	
	//Get EL1904 terminal's MC1 voltage (in mV)
	fbEL2904PriMCmV_ADSRead		: 		ADSREAD ;
	wEL2904_PriMCmV				: 		WORD ;
	xEL2904PriMCmV_busy			: 		BOOL ;
	xEL2904PriMCmV_Err			: 		BOOL ;
	udiEL2904PriMCmV_ErrID		: 		UDINT ;
	
	//Get EL1904 terminal's MC2 voltage (in mV)
	fbEL2904SecMCmV_ADSRead		: 		ADSREAD ;
	wEL2904_SecMCmV				: 		WORD ;
	xEL2904SecMCmV_busy			: 		BOOL ;
	xEL2904SecMCmV_Err			: 		BOOL ;
	udiEL2904SecMCmV_ErrID		: 		UDINT ;

	// EL2904: Error At The Output
	//Bit0-3 is External supply or cross-circuit Error
	//Bit4-7 is Open Load, Current Below 20mA, or Current Above Maximum Value of 500mA
	fbEL2904_OutErr_ADSRead		: 		ADSREAD ;
	wEL2904_OutErr				: 		WORD ;
	xEL2904_OutErr_busy			: 		BOOL ;
	xEL2904_OutErr_Err			: 		BOOL ;
	udiEL2904_OutErr_ErrID		: 		UDINT ;
	
	// EL2904: Supply Error - Field Potential Too High or Too Low
	//Field Voltage from the Power Rail Is Outside The Specification
	fbEL2904_SupplyErr_ADSRead	: 		ADSREAD ;
	wEL2904_SupplyErr			: 		WORD ;
	xEL2904_SupplyErr_busy		: 		BOOL ;
	xEL2904_SupplyErr_Err		: 		BOOL ;
	udiEL2904_SupplyErr_ErrID	: 		UDINT ;

	// EL2904: Temperature Error
	fbEL2904_TempErr_ADSRead	: 		ADSREAD ;
	wEL2904_TempErr				: 		WORD ;
	xEL2904_TempErr_busy		: 		BOOL ;
	xEL2904_TempErr_Err			: 		BOOL ;
	udiEL2904_TempErr_ErrID		: 		UDINT ;

	// EL2904 FEATURES: Standard Output Active/Inactive
	//Standard outputs can be used to directly Enable/Disable a TwinSAFE output
	//if this feature is ACTIVE (Not Turn it ON/OFF, Allow it or not to turn ON!!!)
	fbEL2904_StandardOuts_ADSRead: 		ADSREAD ;
	bEL2904_StandardOuts		: 		BYTE ;
	xEL2904_StandardsOuts_busy	: 		BOOL ;
	xEL2904_StandardsOuts_Err	: 		BOOL ;
	udiEL2904_StandardsOutsID	: 		UDINT ;
	
	// EL2904 FEATURES: Current Measurement Active/Inactive
	//Used to determine TwinSAFE output load current issues
	fbEL2904_CurrMeas_ADSRead	: 		ADSREAD ;
	bEL2904_CurrMeas			: 		BYTE ;
	xEL2904_CurrMeas_busy		: 		BOOL ;
	xEL2904_CurrMeas_Err		: 		BOOL ;
	udiEL2904_CurrMeasID		: 		UDINT ;

	// EL2904 FEATURES: Test Pulses Active/Inactive
	//Used to determine TwinSAFE output wiring is correct
	fbEL2904_TestP_ADSRead		: 		ADSREAD ;
	bEL2904_TestP				: 		BYTE ;
	xEL2904_TestP_busy			: 		BOOL ;
	xEL2904_TestP_Err			: 		BOOL ;
	udiEL2904_TestP_ID			: 		UDINT ;

	// EL2904 FEATURES: Error Acknowledge Active/Inactive
	//Used to reset TwinSAFE output errors instead of focing a cycle power
	//for a TwinSAFE output error
	fbEL2904_ErrAck_ADSRead		: 		ADSREAD;
	bEL2904_ErrAck				: 		BYTE;
	xEL2904_ErrAck_busy			: 		BOOL;
	xEL2904_ErrAck_Err			: 		BOOL;
	udiEL2904_ErrAck_ID			: 		UDINT;
END_VAR
VAR_INPUT
END_VAR

//		8-2-2012
// 		This Program has been supplied by Beckhoff Automation As-Is and is intended only as an example 
//		implementation. Functionality is not guaranteed. 
//
//IF g_bHMI_ScreenBeingDisplayed = 30 THEN
//Interval timer for CoE Reads
T1(
						IN				:= 		NOT xExecute, 
						PT				:=		T#500MS, 
						Q				=>		xExecute, 
						ET				=>		tTime1) ;

C1(
						CU				:= 		xExecute, 
						RESET			:= 		xReset, 
						PV				:= 		wPreset, 
						Q				=> 		xDone, 
						CV				=> 		wCount) ;

IF C1.CV > 6 	THEN xReset := 1 ;
				ELSE xReset := 0 ; 
END_IF ;

// Read the serial number out of the EL2904
fbEL2904Sn_ADSRead(
						NETID			:= 		gc_sADSNetID, 
						PORT			:= 		gc_uiEL2904_EtherCATAdr, 
						IDXGRP			:= 		16#F302, 
						IDXOFFS			:= 		16#F9800002, 
						LEN				:= 		4, 
						DESTADDR		:=		ADR(dwEL2904_Sn), 
						READ			:= 		xExecute, 
						TMOUT			:= 		T#2S, 
						BUSY			=> 		xEL2904Sn_busy, 
						ERR				=> 		xEL2904Sn_Err, 
						ERRID			=> 		xEL2904Sn_ErrID ) ;

g_dwHMI_EL2904Sn 						:= 		dwEL2904_Sn ;

// Read the DIP Switch Setting out of the EL2904
IF C1.CV = 1 THEN
fbEL2904DSw_ADSRead(
						NETID			:= 		gc_sADSNetID, 
						PORT			:= 		gc_uiEL2904_EtherCATAdr, 
						IDXGRP			:= 		16#F302, 
						IDXOFFS			:= 		16#F9800001, 
						LEN				:= 		2, 
						DESTADDR		:=		ADR(wEL2904_DSw), 
						READ			:= 		xExecute, 
						TMOUT			:= 		T#2S, 
						BUSY			=> 		xEL2904DSw_busy, 
						ERR				=> 		xEL2904DSw_Err, 
						ERRID			=> 		udiEL2904DSw_ErrID ) ;

g_wHMI_EL2904DSw 						:= 		wEL2904_DSw ;
END_IF ;

//Read the Hardware Version of the EL2904 Terminal
fbEL2904_HWvers_EcCoESdoRead(
						sNetId			:= 		gc_sADSNetID, 
						nSlaveAddr		:= 		gc_uiEL2904_EtherCATAdr, 
						nSubIndex		:= 		0, 
						nIndex			:= 		16#1009, 
						pDstBuf			:=  	ADR(sEL2904_HWvers),
						cbBufLen		:= 		SIZEOF(sEL2904_HWvers), 
						bExecute		:= 		xExecute, 
						tTimeout		:= 		T#2S, 
						bBusy			=> 		xEL2904_HWvers_Busy, 
						bError			=> 		xEL2904_HWvers_Err, 
						nErrId			=> 		udiEL2904_HWvers_ErrID ) ;

g_sHMI_EL2904_HWvers					:= 		sEL2904_HWvers ;

//Read the Software Version of the EL2904 Logic Terminal (It's f/w)
fbEL2904_FWvers_EcCoESdoRead(
						sNetId			:= 		gc_sADSNetID, 
						nSlaveAddr		:= 		gc_uiEL2904_EtherCATAdr, 
						nSubIndex		:= 		0, 
						nIndex			:= 		16#100A, 
						pDstBuf			:=  	ADR(sEL2904_FWvers),
						cbBufLen		:= 		SIZEOF(sEL2904_FWvers), 
						bExecute		:= 		xExecute, 
						tTimeout		:= 		T#2S, 
						bBusy			=> 		xEL2904_FWvers_Busy, 
						bError			=> 		xEL2904_FWvers_Err, 
						nErrId			=> 		udiEL2904_FWvers_ErrID ) ;

g_sHMI_EL2904_FWvers					:= 		sEL2904_FWvers ;

// EL2904 FEATURES: Standard Output Active/Inactive
//Standard outputs can be used to directly Enable/Disable a TwinSAFE output
//if this feature is ACTIVE (Not Turn it ON/OFF, Allow it or not to turn ON!!!)
IF C1.CV = 0 THEN
fbEL2904_StandardOuts_ADSRead(
						NETID			:= 		gc_sADSNetID, 
						PORT			:= 		gc_uiEL2904_EtherCATAdr, 
						IDXGRP			:= 		16#F302, 
						IDXOFFS			:= 		16#80000001, 
						LEN				:= 		1, 
						DESTADDR		:=		ADR(bEL2904_StandardOuts), 
						READ			:= 		xExecute, 
						TMOUT			:= 		T#2S, 
						BUSY			=> 		xEL2904_StandardsOuts_busy, 
						ERR				=> 		xEL2904_StandardsOuts_Err, 
						ERRID			=> 		udiEL2904_StandardsOutsID );

g_xHMI_EL2904_StandardOuts				:= 		bEL2904_StandardOuts.0 ;
END_IF ;

//EL2904 FEATURES: Current Measurement Active/Inactive
//Used to determine TwinSAFE output load current issues
IF C1.CV = 2 THEN
fbEL2904_CurrMeas_ADSRead(
						NETID			:= 		gc_sADSNetID, 
						PORT			:= 		gc_uiEL2904_EtherCATAdr, 
						IDXGRP			:= 		16#F302, 
						IDXOFFS			:= 		16#80000002, 
						LEN				:= 		1, 
						DESTADDR		:=		ADR(bEL2904_CurrMeas), 
						READ			:= 		xExecute, 
						TMOUT			:= 		T#2S, 
						BUSY			=> 		xEL2904_CurrMeas_busy, 
						ERR				=> 		xEL2904_CurrMeas_Err, 
						ERRID			=> 		udiEL2904_CurrMeasID );

g_xHMI_EL2904_CurrentMeas				:= 		bEL2904_CurrMeas.0 ;
END_IF ;

//EL2904 FEATURES: Test Pulses Active/Inactive
//Used to determine TwinSAFE output wiring is correct
IF C1.CV = 4 THEN
fbEL2904_TestP_ADSRead(
						NETID			:= 		gc_sADSNetID, 
						PORT			:= 		gc_uiEL2904_EtherCATAdr, 
						IDXGRP			:= 		16#F302, 
						IDXOFFS			:= 		16#80000003, 
						LEN				:= 		1, 
						DESTADDR		:=		ADR(bEL2904_TestP), 
						READ			:= 		xExecute, 
						TMOUT			:= 		T#2S, 
						BUSY			=> 		xEL2904_TestP_busy, 
						ERR				=> 		xEL2904_TestP_Err, 
						ERRID			=> 		udiEL2904_TestP_ID );

g_xHMI_EL2904_TestPulses				:= 		bEL2904_TestP.0 ;
END_IF ;

//EL2904 FEATURES: Error Acknowledge Active/Inactive
//Used to reset TwinSAFE output errors instead of forcing a cycle power
//for a TwinSAFE output error
IF C1.CV = 6 THEN
fbEL2904_ErrAck_ADSRead(
						NETID			:= 		gc_sADSNetID, 
						PORT			:= 		gc_uiEL2904_EtherCATAdr, 
						IDXGRP			:= 		16#F302, 
						IDXOFFS			:= 		16#80000004, 
						LEN				:= 		1, 
						DESTADDR		:= 		ADR(bEL2904_ErrAck), 
						READ			:= 		xExecute, 
						TMOUT			:= 		T#2S, 
						BUSY			=> 		xEL2904_ErrAck_busy, 
						ERR				=> 		xEL2904_ErrAck_Err, 
						ERRID			=> 		udiEL2904_ErrAck_ID );
						

g_xHMI_EL2904_ErrAck					:= 		bEL2904_ErrAck.0 ;
END_IF ;

// Read the Primary Micro Controller (MC1) Temperature in DegC out of the EL2904
IF C1.CV = 2 THEN
fbEL2904PriMCTemp_ADSRead(
						NETID			:= 		gc_sADSNetID, 
						PORT			:= 		gc_uiEL2904_EtherCATAdr, 
						IDXGRP			:= 		16#F302, 
						IDXOFFS			:= 		16#FA800001, 
						LEN				:= 		2, 
						DESTADDR		:=		ADR(wEL2904_PriMCTemp), 
						READ			:= 		xExecute, 
						TMOUT			:= 		T#2S, 
						BUSY			=> 		xEL2904PriMCTemp_busy, 
						ERR				=> 		xEL2904PriMCTemp_Err, 
						ERRID			=> 		udiEL2904PriMCTemp_ErrID );

g_wHMI_EL2904PriMCTemp 					:= 		wEL2904_PriMCTemp ;
END_IF ;

// Read the Secondary Micro Controller (MC2) Temperature in DegC out of the EL2904
IF C1.CV = 2 THEN
fbEL2904SecMCTemp_ADSRead(
						NETID			:= 		gc_sADSNetID, 
						PORT			:= 		gc_uiEL2904_EtherCATAdr, 
						IDXGRP			:= 		16#F302, 
						IDXOFFS			:= 		16#FA800002, 
						LEN				:= 		2, 
						DESTADDR		:=		ADR(wEL2904_SecMCTemp), 
						READ			:= 		xExecute, 
						TMOUT			:= 		T#2S, 
						BUSY			=> 		xEL2904SecMCTemp_busy, 
						ERR				=> 		xEL2904SecMCTemp_Err, 
						ERRID			=> 		udiEL2904SecMCTemp_ErrID );

g_wHMI_EL2904SecMCTemp 					:= 		wEL2904_SecMCTemp ;
END_IF ;

// Read the Primary Micro Controller (MC1) Voltage in mV out of the EL2904
IF C1.CV = 3 THEN
fbEL2904PriMCmV_ADSRead(
						NETID			:= 		gc_sADSNetID, 
						PORT			:= 		gc_uiEL2904_EtherCATAdr, 
						IDXGRP			:= 		16#F302, 
						IDXOFFS			:= 		16#FA810001, 
						LEN				:= 		2, 
						DESTADDR		:=		ADR(wEL2904_PriMCmV), 
						READ			:= 		xExecute, 
						TMOUT			:= 		T#2S, 
						BUSY			=> 		xEL2904PriMCmV_busy, 
						ERR				=> 		xEL2904PriMCmV_Err, 
						ERRID			=> 		udiEL2904PriMCmV_ErrID );
						
g_wHMI_EL2904PriMC_Volts				:= 		WORD_TO_LREAL(wEL2904_PriMCmV) / 1000.0 ;
END_IF ;

// Read the Secondary Micro Controller (MC2) Voltage in mV out of the EL2904
IF C1.CV = 3 THEN
fbEL2904SecMCmV_ADSRead(
						NETID			:= 		gc_sADSNetID, 
						PORT			:= 		gc_uiEL2904_EtherCATAdr, 
						IDXGRP			:= 		16#F302, 
						IDXOFFS			:= 		16#FA810002, 
						LEN				:= 		2, 
						DESTADDR		:=		ADR(wEL2904_SecMCmV), 
						READ			:= 		xExecute, 
						TMOUT			:= 		T#2S, 
						BUSY			=> 		xEL2904SecMCmV_busy, 
						ERR				=> 		xEL2904SecMCmV_Err, 
						ERRID			=> 		udiEL2904SecMCmV_ErrID );
						
g_wHMI_EL2904SecMC_Volts 				:= 		WORD_TO_LREAL(wEL2904_SecMCmV) / 1000.0 ;
END_IF ;
//	ELSE xReset := 1 ;
//	END_IF ;
//	
//	EL2904 ALARMS
//
//EL2904: Error At The Output
//Bit0-3 is External supply or cross-circuit Error
//Bit4-7 is Open Load, Current Below 20mA, or Current Above Maximum Value of 500mA
fbEL2904_OutErr_ADSRead(
						NETID			:= 		gc_sADSNetID, 
						PORT			:= 		gc_uiEL2904_EtherCATAdr, 
						IDXGRP			:= 		16#F302, 
						IDXOFFS			:= 		16#800E000C, 
						LEN				:= 		2, 
						DESTADDR		:=		ADR(wEL2904_OutErr), 
						READ			:= 		xExecute, 
						TMOUT			:= 		T#2S, 
						BUSY			=> 		xEL2904_OutErr_busy, 
						ERR				=> 		xEL2904_OutErr_Err, 
						ERRID			=> 		udiEL2904_OutErr_ErrID );

//These errors may only be present temporarily so they need to be latched and then cleared
//to be properly noted by the operator
g_xHMI_EL2904_ExtSup_CrossCirErr_Out1	:= 		wEL2904_OutErr.0 OR (g_xHMI_EL2904_ExtSup_CrossCirErr_Out1 AND NOT g_xHMI_EL2904_ErrClearPB) ;
g_xHMI_EL2904_ExtSup_CrossCirErr_Out2	:= 		wEL2904_OutErr.1 OR (g_xHMI_EL2904_ExtSup_CrossCirErr_Out2 AND NOT g_xHMI_EL2904_ErrClearPB) ;
g_xHMI_EL2904_ExtSup_CrossCirErr_Out3	:= 		wEL2904_OutErr.2 OR (g_xHMI_EL2904_ExtSup_CrossCirErr_Out3 AND NOT g_xHMI_EL2904_ErrClearPB) ;
g_xHMI_EL2904_ExtSup_CrossCirErr_Out4	:= 		wEL2904_OutErr.3 OR (g_xHMI_EL2904_ExtSup_CrossCirErr_Out4 AND NOT g_xHMI_EL2904_ErrClearPB) ;
g_xHMI_EL2904_OutLoadErr_Out1			:= 		wEL2904_OutErr.4 OR (g_xHMI_EL2904_OutLoadErr_Out1 AND NOT g_xHMI_EL2904_ErrClearPB) ;
g_xHMI_EL2904_OutLoadErr_Out2			:= 		wEL2904_OutErr.5 OR (g_xHMI_EL2904_OutLoadErr_Out2 AND NOT g_xHMI_EL2904_ErrClearPB) ;
g_xHMI_EL2904_OutLoadErr_Out3			:= 		wEL2904_OutErr.6 OR (g_xHMI_EL2904_OutLoadErr_Out3 AND NOT g_xHMI_EL2904_ErrClearPB) ;
g_xHMI_EL2904_OutLoadErr_Out4			:= 		wEL2904_OutErr.7 OR (g_xHMI_EL2904_OutLoadErr_Out4 AND NOT g_xHMI_EL2904_ErrClearPB) ;


//EL2904: Power Rail Supply Error - Field Potential Too High or Too Low
//Field Voltage from the Power Rail Is Outside The Specification
//Documentation says this is in 800E:0D but testing shows it's in 800E:0A
//Value = 0x1101 when voltage is below 17.4 v
//Value = 0x1110 when voltage is above 20.8 v
fbEL2904_SupplyErr_ADSRead(
						NETID			:= 		gc_sADSNetID, 
						PORT			:= 		gc_uiEL2904_EtherCATAdr, 
						IDXGRP			:= 		16#F302, 
						IDXOFFS			:= 		16#800E000A, 
						LEN				:= 		2, 
						DESTADDR		:=		ADR(wEL2904_SupplyErr), 
						READ			:= 		xExecute, 
						TMOUT			:= 		T#2S, 
						BUSY			=> 		xEL2904_SupplyErr_busy, 
						ERR				=> 		xEL2904_SupplyErr_Err, 
						ERRID			=> 		udiEL2904_SupplyErr_ErrID );

//These errors may only be present temporarily so they need to be latched and then cleared
//to be properly noted by the operator
g_xHMI_EL2904_PwrRailVoltageHi			:= 		(NOT wEL2904_SupplyErr.0 AND wEL2904_SupplyErr.1 AND wEL2904_SupplyErr.2 AND wEL2904_SupplyErr.3) OR (g_xHMI_EL2904_PwrRailVoltageHi AND NOT g_xHMI_EL2904_ErrClearPB) ;
g_xHMI_EL2904_PwrRailVoltageLo			:= 		(wEL2904_SupplyErr.0 AND wEL2904_SupplyErr.1 AND NOT wEL2904_SupplyErr.2 AND wEL2904_SupplyErr.3) OR (g_xHMI_EL2904_PwrRailVoltageLo AND NOT g_xHMI_EL2904_ErrClearPB) ;


//EL2904: Temperature Error
//There are two temperature sensors inside each Microcontroller and another
//on the Output Circuit Board
fbEL2904_TempErr_ADSRead(
						NETID			:= 		gc_sADSNetID, 
						PORT			:= 		gc_uiEL2904_EtherCATAdr, 
						IDXGRP			:= 		16#F302, 
						IDXOFFS			:= 		16#800E000E, 
						LEN				:= 		2, 
						DESTADDR		:=		ADR(wEL2904_TempErr), 
						READ			:= 		xExecute, 
						TMOUT			:= 		T#2S, 
						BUSY			=> 		xEL2904_TempErr_busy, 
						ERR				=> 		xEL2904_TempErr_Err, 
						ERRID			=> 		udiEL2904_TempErr_ErrID );

//These errors may only be present temporarily so they need to be latched and then cleared
//to be properly noted by the operator
g_xHMI_EL2904_TempErr_OTMc1				:= 		wEL2904_TempErr.0 OR (g_xHMI_EL2904_TempErr_OTMc1 AND NOT g_xHMI_EL2904_ErrClearPB) ;
g_xHMI_EL2904_TempErr_OTMc2				:= 		wEL2904_TempErr.1 OR (g_xHMI_EL2904_TempErr_OTMc2 AND NOT g_xHMI_EL2904_ErrClearPB) ;
g_xHMI_EL2904_TempErr_OTOutBoard		:= 		wEL2904_TempErr.2 OR (g_xHMI_EL2904_TempErr_OTOutBoard AND NOT g_xHMI_EL2904_ErrClearPB) ;
g_xHMI_EL2904_TempErr_UTMc1				:= 		wEL2904_TempErr.3 OR (g_xHMI_EL2904_TempErr_UTMc1 AND NOT g_xHMI_EL2904_ErrClearPB) ;
g_xHMI_EL2904_TempErr_UTMc2				:= 		wEL2904_TempErr.4 OR (g_xHMI_EL2904_TempErr_UTMc2 AND NOT g_xHMI_EL2904_ErrClearPB) ;
g_xHMI_EL2904_TempErr_UTOutBoard		:= 		wEL2904_TempErr.5 OR (g_xHMI_EL2904_TempErr_UTOutBoard AND NOT g_xHMI_EL2904_ErrClearPB) ;
g_xHMI_EL2904_TempErr_DiffOnBoard		:= 		wEL2904_TempErr.6 OR (g_xHMI_EL2904_TempErr_DiffOnBoard AND NOT g_xHMI_EL2904_ErrClearPB) ;
g_xHMI_EL2904_TempErr_DiffBetweenMc1Mc2	:= 		wEL2904_TempErr.7 OR (g_xHMI_EL2904_TempErr_DiffBetweenMc1Mc2 AND NOT g_xHMI_EL2904_ErrClearPB) ;


//Sum of all errors we know of in the EL2904 terminal
IF 		g_xHMI_EL2904_ExtSup_CrossCirErr_Out1 
	OR 	g_xHMI_EL2904_ExtSup_CrossCirErr_Out2
	OR 	g_xHMI_EL2904_ExtSup_CrossCirErr_Out3 
	OR 	g_xHMI_EL2904_ExtSup_CrossCirErr_Out4
	OR 	g_xHMI_EL2904_OutLoadErr_Out1
	OR 	g_xHMI_EL2904_OutLoadErr_Out2
	OR 	g_xHMI_EL2904_OutLoadErr_Out3
	OR 	g_xHMI_EL2904_OutLoadErr_Out4
	OR	g_xHMI_EL2904_PwrRailVoltageHi
	OR	g_xHMI_EL2904_PwrRailVoltageLo
	OR	g_xHMI_EL2904_TempErr_OTMc1
	OR	g_xHMI_EL2904_TempErr_OTMc2
	OR	g_xHMI_EL2904_TempErr_OTOutBoard
	OR	g_xHMI_EL2904_TempErr_UTMc1
	OR	g_xHMI_EL2904_TempErr_UTMc2
	OR	g_xHMI_EL2904_TempErr_UTOutBoard
	OR	g_xHMI_EL2904_TempErr_DiffOnBoard
	OR	g_xHMI_EL2904_TempErr_DiffBetweenMc1Mc2
		THEN g_xHMI_EL2904_General_Error := TRUE ;
		ELSE g_xHMI_EL2904_General_Error := FALSE ;
END_IF ;

END_PROGRAM

// ---- POUs/Safety_Diagnostics/AX5805_ADS_Reads.TcPOU
PROGRAM AX5805_ADS_Reads
//		8-2-2012
// 		This Program has been supplied by Beckhoff Automation As-Is and is intended only as an example 
//		implementation. Functionality is not guaranteed. 
//
VAR
	//Time to check CoE values
	T1							: 		TON ;
	xExecute					: 		BOOL ;
	tTime1						: 		TIME ;

	//Counter for just some very simple sequencing
	C1							: 		CTU ;
	xReset						: 		BOOL ;
	wPreset						: 		WORD := 10 ;
	xDone						: 		BOOL ;
	wCount						: 		WORD ;

	// Reading the serial number out of the AX5805
	fbAX5805Sn_ADSRead			: 		ADSREAD ;
	dwAX5805_Sn					: 		DWORD ;
	xAX5805Sn_busy				: 		BOOL ;
	xAX5805Sn_Err				: 		BOOL ;
	xAX5805Sn_ErrID				: 		UDINT ;

	// Reading the DIP Switch Setting out of the AX5805
	fbAX5805DSw_ADSRead			: 		ADSREAD ;
	wAX5805_DSw					: 		WORD ;
	xAX5805DSw_busy				: 		BOOL ;
	xAX5805DSw_Err				: 		BOOL ;
	udiAX5805DSw_ErrID			: 		UDINT ;

	//Read the Hardware Version of the AX5805 Logic Terminal
	fbAX5805_HWvers_EcCoESdoRead: 		FB_EcCoESdoRead ;
	sAX5805_HWvers				: 		STRING(2) ;
	xAX5805_HWvers_Busy			: 		BOOL ;
	xAX5805_HWvers_Err			: 		BOOL ;
	udiAX5805_HWvers_ErrID		: 		UDINT ;

	//Read the Software Version of the AX5805 Logic Terminal (It's f/w)
	fbAX5805_FWvers_EcCoESdoRead: 		FB_EcCoESdoRead ;
	sAX5805_FWvers				: 		STRING(2) ;
	xAX5805_FWvers_Busy			: 		BOOL ;
	xAX5805_FWvers_Err			: 		BOOL ;
	udiAX5805_FWvers_ErrID		: 		UDINT ;

	//Read the Number Of Connections Configured In The AX5805 Logic Terminal
	fbAX5805_StatConn_EcCoESdoRead: 	FB_EcCoESdoRead ;
	bAX5805_NoOfConnections		: 		BYTE ;
	xAX5805_NoOfConnections_Busy: 		BOOL ;
	xAX5805_NoOfConnections_Err	: 		BOOL ;
	udiAX5805_NoOfConnections_ErrID: 	UDINT ;

	//Read the Number Of Safety Groups Configured In The AX5805 Logic Terminal
	fbAX5805_SafetyGrps_EcCoESdoRead: 	FB_EcCoESdoRead ;
	bAX5805_NoOfSafetyGrps		: 		BYTE ;
	xAX5805_NoOfSafetyGrps_Busy	: 		BOOL ;
	xAX5805_NoOfSafetyGrps_Err	: 		BOOL ;
	udiAX5805_NoOfSafetyGrps_ErrID: 	UDINT ;

	//Read the Number Of Safety Function Blocks Configured In The AX5805 Logic Terminal
	fbAX5805_SafetyFBs_EcCoESdoRead: 	FB_EcCoESdoRead ;
	bAX5805_NoOfSafetyFBs		: 		BYTE ;
	xAX5805_NoOfSafetyFBs_Busy	: 		BOOL ;
	xAX5805_NoOfSafetyFBs_Err	: 		BOOL ;
	udiAX5805_NoOfSafetyFBs_ErrID: 		UDINT ;
	
	// Reading the Primary Micro Controller (MC1) Temperature in DegC out of the AX5805
	fbAX5805PriMCTemp_ADSRead	: 		ADSREAD ;
	wAX5805_PriMCTemp			: 		WORD ;
	xAX5805PriMCTemp_busy		: 		BOOL ;
	xAX5805PriMCTemp_Err		: 		BOOL ;
	udiAX5805PriMCTemp_ErrID	: 		UDINT ;

	// Reading the Secondary Micro Controller (MC2) Temperature in DegC out of the AX5805
	fbAX5805SecMCTemp_ADSRead	: 		ADSREAD ;
	wAX5805_SecMCTemp			: 		WORD ;
	xAX5805SecMCTemp_busy		: 		BOOL ;
	xAX5805SecMCTemp_Err		: 		BOOL ;
	udiAX5805SecMCTemp_ErrID	: 		UDINT ;

	// Reading the Primary Micro Controller (MC1) Voltage in mV out of the AX5805
	fbAX5805PriMC3300mV_ADSRead	: 		ADSREAD ;
	wAX5805_PriMC3300mV			: 		WORD ;
	xAX5805PriMC3300mV_busy		: 		BOOL ;
	xAX5805PriMC3300mV_Err		: 		BOOL ;
	udiAX5805PriMC3300mV_ErrID	: 		UDINT ;
	fbAX5805PriMC5000mV_ADSRead	: 		ADSREAD ;
	wAX5805_PriMC5000mV			: 		WORD ;
	xAX5805PriMC5000mV_busy		: 		BOOL ;
	xAX5805PriMC5000mV_Err		: 		BOOL ;
	udiAX5805PriMC5000mV_ErrID	: 		UDINT ;
	
	// Reading the Secondary Micro Controller (MC2) Voltage in mV out of the AX5805
	fbAX5805SecMC3300mV_ADSRead	: 		ADSREAD ;
	wAX5805_SecMC3300mV			: 		WORD ;
	xAX5805SecMC3300mV_busy		: 		BOOL ;
	xAX5805SecMC3300mV_Err		: 		BOOL ;
	udiAX5805SecMC3300mV_ErrID	: 		UDINT ;
	fbAX5805SecMC5000mV_ADSRead	: 		ADSREAD ;
	wAX5805_SecMC5000mV			: 		WORD ;
	xAX5805SecMC5000mV_busy		: 		BOOL ;
	xAX5805SecMC5000mV_Err		: 		BOOL ;
	udiAX5805SecMC5000mV_ErrID	: 		UDINT ;

	//Read the Configured Safety Option In The AX5000 Drive
	fbAX5000_SafetyOption				: 		FB_SoERead ;
	dwSafetyOption						: 		DWORD ;
	Axis1 								: 		AXIS_REF ;
	xAX5000_SafetyOption_busy			: 		BOOL ;
	xAX5000_SafetyOption_Err			: 		BOOL ;
	udiAX5000_SafetyOption_ErrID		: 		UDINT ;
	uiAX5000_SafetyOption_SercosErrID	: 		UINT ;
	dwAX5000_SafetyOption_Attribute		: 		DWORD ;
	
	//Read the Configured Motor String For CH-A in The AX5000 Drive
	fbAX5000_ConfigMotorCHA				: 		FB_SoERead ;
	sConfigMotorCHA						: 		STRING(30) ;
	xAX5000_sConfigMotorCHA_busy		: 		BOOL ;
	xAX5000_sConfigMotorCHA_Err			: 		BOOL ;
	udiAX5000_sConfigMotorCHA_ErrID		: 		UINT ;
	xAX5000_ConfigMotorCHA_busy			: 		BOOL ;
	xAX5000_ConfigMotorCHA_Err			:		BOOL ;
	udiAX5000_ConfigMotorCHA_ErrID		: 		UDINT ;
	uiAX5000_ConfigMotorCHA_SercosErrID	: 		UINT ;
	dwAX5000_ConfigMotorCHA_Attribute	: 		DWORD ;
	ConfigMotorCHA						: 		ARRAY[0..29] OF UINT ;
END_VAR
VAR_INPUT
END_VAR

//		8-2-2012
// 		This Program has been supplied by Beckhoff Automation As-Is and is intended only as an example 
//		implementation. Functionality is not guaranteed. 
//
IF g_bHMI_ScreenBeingDisplayed = 60 THEN
// Interval timer for CoE Reads
T1(
						IN				:= 		NOT xExecute, 
						PT				:=		T#500MS, 
						Q				=>		xExecute, 
						ET				=>		tTime1 ) ;

C1(
						CU				:= 		xExecute, 
						RESET			:= 		xReset, 
						PV				:= 		wPreset, 
						Q				=> 		xDone, 
						CV				=> 		wCount) ;

IF C1.CV > 6 	THEN xReset := 1 ;
				ELSE xReset := 0 ; 
END_IF ;

// Read the serial number out of the AX5805
fbAX5805Sn_ADSRead(
						NETID			:= 		gc_sADSNetID, 
						PORT			:= 		gc_uiAX5805_EtherCATAdr, 
						IDXGRP			:= 		16#F302, 
						IDXOFFS			:= 		16#F9800002, 
						LEN				:= 		4, 
						DESTADDR		:= 		ADR(dwAX5805_Sn), 
						READ			:= 		xExecute, 
						TMOUT			:= 		T#2S, 
						BUSY			=> 		xAX5805Sn_busy, 
						ERR				=> 		xAX5805Sn_Err, 
						ERRID			=> 		xAX5805Sn_ErrID );

g_dwHMI_AX5805Sn 						:= 		dwAX5805_Sn ;

// Read the DIP Switch Setting out of the AX5805
IF C1.CV = 1 THEN
fbAX5805DSw_ADSRead(
						NETID			:= 		gc_sADSNetID, 
						PORT			:= 		gc_uiAX5805_EtherCATAdr, 
						IDXGRP			:= 		16#F302, 
						IDXOFFS			:= 		16#F9800001, 
						LEN				:= 		2, 
						DESTADDR		:= 		ADR(wAX5805_DSw), 
						READ			:= 		xExecute, 
						TMOUT			:= 		T#2S, 
						BUSY			=> 		xAX5805DSw_busy, 
						ERR				=> 		xAX5805DSw_Err, 
						ERRID			=> 		udiAX5805DSw_ErrID );

g_wHMI_AX5805DSw 						:= 		wAX5805_DSw ;
END_IF ;						

//Read the Hardware Version of the AX5805 Logic Terminal
fbAX5805_HWvers_EcCoESdoRead(
						sNetId			:= 		gc_sADSNetID, 
						nSlaveAddr		:= 		gc_uiAX5805_EtherCATAdr, 
						nSubIndex		:= 		0, 
						nIndex			:= 		16#1009, 
						pDstBuf			:=  	ADR(sAX5805_HWvers),
						cbBufLen		:= 		SIZEOF(sAX5805_HWvers), 
						bExecute		:= 		xExecute, 
						tTimeout		:= 		T#2S, 
						bBusy			=> 		xAX5805_HWvers_Busy, 
						bError			=> 		xAX5805_HWvers_Err, 
						nErrId			=> 		udiAX5805_HWvers_ErrID ) ;

g_sHMI_AX5805_HWvers					:= 		sAX5805_HWvers ;

//Read the Software Version of the AX5805 Logic Terminal (It's f/w)
fbAX5805_FWvers_EcCoESdoRead(
						sNetId			:= 		gc_sADSNetID, 
						nSlaveAddr		:= 		gc_uiAX5805_EtherCATAdr, 
						nSubIndex		:= 		0, 
						nIndex			:= 		16#100A, 
						pDstBuf			:=  	ADR(sAX5805_FWvers),
						cbBufLen		:= 		SIZEOF(sAX5805_FWvers), 
						bExecute		:= 		xExecute, 
						tTimeout		:= 		T#2S, 
						bBusy			=> 		xAX5805_FWvers_Busy, 
						bError			=> 		xAX5805_FWvers_Err, 
						nErrId			=> 		udiAX5805_FWvers_ErrID ) ;

g_sHMI_AX5805_FWvers					:= 		sAX5805_FWvers ;

// Read the Primary Micro Controller (MC1) Temperature in DegC out of the AX5805
IF C1.CV = 2 THEN
fbAX5805PriMCTemp_ADSRead(
						NETID			:= 		gc_sADSNetID, 
						PORT			:= 		gc_uiAX5805_EtherCATAdr, 
						IDXGRP			:= 		16#F302, 
						IDXOFFS			:= 		16#FA800001, 
						LEN				:= 		2, 
						DESTADDR		:= 		ADR(wAX5805_PriMCTemp), 
						READ			:= 		xExecute, 
						TMOUT			:= 		T#2S, 
						BUSY			=> 		xAX5805PriMCTemp_busy, 
						ERR				=> 		xAX5805PriMCTemp_Err, 
						ERRID			=> 		udiAX5805PriMCTemp_ErrID );

g_wHMI_AX5805PriMCTemp 					:= 		wAX5805_PriMCTemp ;
END_IF ;

// Read the Secondary Micro Controller (MC2) Temperature in DegC out of the AX5805
IF C1.CV = 3 THEN
fbAX5805SecMCTemp_ADSRead(
						NETID			:= 		gc_sADSNetID, 
						PORT			:= 		gc_uiAX5805_EtherCATAdr, 
						IDXGRP			:= 		16#F302, 
						IDXOFFS			:= 		16#FA800002, 
						LEN				:= 		2, 
						DESTADDR		:= 		ADR(wAX5805_SecMCTemp), 
						READ			:= 		xExecute, 
						TMOUT			:= 		T#2S, 
						BUSY			=> 		xAX5805SecMCTemp_busy, 
						ERR				=> 		xAX5805SecMCTemp_Err, 
						ERRID			=> 		udiAX5805SecMCTemp_ErrID );

g_wHMI_AX5805SecMCTemp 					:= 		wAX5805_SecMCTemp ;
END_IF ;

// Read the Primary Micro Controller (MC1) 3.3v Nominal Voltage in mV out of the AX5805
IF C1.CV = 4 THEN
fbAX5805PriMC3300mV_ADSRead(
						NETID			:= 		gc_sADSNetID, 
						PORT			:= 		gc_uiAX5805_EtherCATAdr, 
						IDXGRP			:= 		16#F302, 
						IDXOFFS			:= 		16#FA810001, 
						LEN				:= 		2, 
						DESTADDR		:= 		ADR(wAX5805_PriMC3300mV), 
						READ			:= 		xExecute, 
						TMOUT			:= 		T#2S, 
						BUSY			=> 		xAX5805PriMC3300mV_busy, 
						ERR				=> 		xAX5805PriMC3300mV_Err, 
						ERRID			=> 		udiAX5805PriMC3300mV_ErrID );

g_wHMI_AX5805PriMC_3p3Volts				:= 		WORD_TO_LREAL(wAX5805_PriMC3300mV) / 1000.0 ;
END_IF ;

// Read the Secondary Micro Controller (MC2) 3.3v Nominal Voltage in mV out of the AX5805
IF C1.CV = 5 THEN
fbAX5805SecMC3300mV_ADSRead(
						NETID			:= 		gc_sADSNetID, 
						PORT			:= 		gc_uiAX5805_EtherCATAdr, 
						IDXGRP			:= 		16#F302, 
						IDXOFFS			:= 		16#FA810002, 
						LEN				:= 		2, 
						DESTADDR		:= 		ADR(wAX5805_SecMC3300mV), 
						READ			:= 		xExecute, 
						TMOUT			:= 		T#2S, 
						BUSY			=> 		xAX5805SecMC3300mV_busy, 
						ERR				=> 		xAX5805SecMC3300mV_Err, 
						ERRID			=> 		udiAX5805SecMC3300mV_ErrID );
			
g_wHMI_AX5805SecMC_3p3Volts 				:= 		WORD_TO_LREAL(wAX5805_SecMC3300mV) / 1000.0 ;
END_IF ;

// Read the Primary Micro Controller (MC1) 5.0v Nominal Voltage in mV out of the AX5805
IF C1.CV = 1 THEN
fbAX5805PriMC5000mV_ADSRead(
						NETID			:= 		gc_sADSNetID, 
						PORT			:= 		gc_uiAX5805_EtherCATAdr, 
						IDXGRP			:= 		16#F302, 
						IDXOFFS			:= 		16#FA810003, 
						LEN				:= 		2, 
						DESTADDR		:= 		ADR(wAX5805_PriMC5000mV), 
						READ			:= 		xExecute, 
						TMOUT			:= 		T#2S, 
						BUSY			=> 		xAX5805PriMC5000mV_busy, 
						ERR				=> 		xAX5805PriMC5000mV_Err, 
						ERRID			=> 		udiAX5805PriMC5000mV_ErrID );

g_wHMI_AX5805PriMC_5Volts				:= 		WORD_TO_LREAL(wAX5805_PriMC5000mV) / 1000.0 ;
END_IF ;

// Read the Secondary Micro Controller (MC2) 5.0v Nominal Voltage in mV out of the AX5805
IF C1.CV = 2 THEN
fbAX5805SecMC5000mV_ADSRead(
						NETID			:= 		gc_sADSNetID, 
						PORT			:= 		gc_uiAX5805_EtherCATAdr, 
						IDXGRP			:= 		16#F302, 
						IDXOFFS			:= 		16#FA810004, 
						LEN				:= 		2, 
						DESTADDR		:= 		ADR(wAX5805_SecMC5000mV), 
						READ			:= 		xExecute, 
						TMOUT			:= 		T#2S, 
						BUSY			=> 		xAX5805SecMC5000mV_busy, 
						ERR				=> 		xAX5805SecMC5000mV_Err, 
						ERRID			=> 		udiAX5805SecMC5000mV_ErrID );
			
g_wHMI_AX5805SecMC_5Volts 				:= 		WORD_TO_LREAL(wAX5805_SecMC5000mV) / 1000.0 ;
END_IF ;

(* Read the Configured Safety Option For CH-A in The AX5000 Drive

An advantage of using the FB_SoERead function block Form the MC2_Drive library
is the NedID is the controller's NetID not the EtherCAT master so it is possible 
to leave that field with just blank single quotes '' and the TwinCAT system 
assumes the NetID of the computer for you.

The MC2_Drive library has dependencies on the MC2 library in TwinCAT and Tc3 at this point
(build 3099.1) doesn't notice the dependancy and add the extra library for you.  You must
manually add it yourself.

	S_0_IDN		: WORD	:= 16#0000;
	S_1_IDN		: WORD	:= 16#1000;
	S_2_IDN		: WORD	:= 16#2000;
	S_3_IDN		: WORD	:= 16#3000;
	S_4_IDN		: WORD	:= 16#4000;
	S_5_IDN		: WORD	:= 16#5000;
	S_6_IDN		: WORD	:= 16#6000;
	S_7_IDN		: WORD	:= 16#7000;

	P_0_IDN		: WORD	:= 16#8000;
	P_1_IDN		: WORD	:= 16#9000;
	P_2_IDN		: WORD	:= 16#A000;
	P_3_IDN		: WORD	:= 16#B000;
	P_4_IDN		: WORD	:= 16#C000;
	P_5_IDN		: WORD	:= 16#D000;
	P_6_IDN		: WORD	:= 16#E000;
	P_7_IDN		: WORD	:= 16#F000;

A Few documented SERCOS error codes:
---------------------------------------
0x1003 Wrong parameter mode 
0x1004 Data parameter wrong value size 
0x1005 False backup parameter type  
0x1006 Backup list was not IDN 192 

nElement: Element number of the parameter that is to be written. The following values are allowed:
--------------------------------------------------------------------------------------------------
Value Description 
0x01 Data Status 
0x02 Name (read only) 
0x04 Attribute 
0x08 Unit 
0x10 Minimum 
0x20 Maximum 
0x40 Value 
0x80 Default 

*)
fbAX5000_SafetyOption(
						NetId			:= 		'', 
						Idn				:= 		DINT_TO_WORD(16#8000 + 2000), 
						Element			:= 		16#40, 
						pDstBuf			:= 		ADR(dwSafetyOption), 
						BufLen			:= 		SIZEOF(dwSafetyOption), 
						Execute			:= 		xExecute, 
						Timeout			:= 		T#2S, 
						Axis			:= 		Axis1, 
						Busy			=> 		xAX5000_SafetyOption_busy, 
						Error			=> 		xAX5000_SafetyOption_Err, 
						AdsErrId		=> 		udiAX5000_SafetyOption_ErrID, 
						SercosErrId		=> 		uiAX5000_SafetyOption_SercosErrID, 
						Attribute		=> 		dwAX5000_SafetyOption_Attribute) ;

IF dwSafetyOption 						= 		0 THEN
	g_sHMI_AX5000_SafetyOption			:= 		'No Safety Option Selected' ;
	ELSIF dwSafetyOption				= 		1 THEN
	g_sHMI_AX5000_SafetyOption			:= 		'AX5801 Option Selected' ;
	ELSIF dwSafetyOption				= 		2 THEN
	g_sHMI_AX5000_SafetyOption			:= 		'AX5805 Option Selected' ;
ELSE
	g_sHMI_AX5000_SafetyOption			:= 		'Invalid Option' ;
END_IF ;

//AX5000 Ch-A Motor String
fbAX5000_ConfigMotorCHA(
						NetId			:= 		'', 
						Idn				:= 		DINT_TO_WORD(16#8000 + 53), 
						Element			:= 		16#40, 
						pDstBuf			:= 		ADR(ConfigMotorCHA), 
						BufLen			:= 		SIZEOF(ConfigMotorCHA), 
						Execute			:= 		xExecute, 
						Timeout			:= 		T#2S, 
						Axis			:= 		Axis1, 
						Busy			=> 		xAX5000_ConfigMotorCHA_busy, 
						Error			=> 		xAX5000_ConfigMotorCHA_Err, 
						AdsErrId		=> 		udiAX5000_ConfigMotorCHA_ErrID, 
						SercosErrId		=> 		uiAX5000_ConfigMotorCHA_SercosErrID, 
						Attribute		=> 		dwAX5000_ConfigMotorCHA_Attribute) ;

g_sHMI_AX5000_ConfigMotorCHA 			:= 		 UINT_TO_STRING(ConfigMotorCHA[2]) ;

ELSE xReset := 1 ;
END_IF ;

END_PROGRAM

// ---- POUs/TwinSAFE_Function_Blocks_Info/FB_InfoConnectionShutdown.TcPOU
FUNCTION_BLOCK FB_InfoConnectionShutdown
VAR_INPUT
	stInfoData 		: 		DUT_ST_InfoDataFB ;
END_VAR
VAR_OUTPUT
	sState 			: 		STRING ;
	sDiag  			: 		STRING ;
END_VAR
VAR
END_VAR

// Connection Shutdown FB's State
IF stInfoData.usiMapState 			= 	0 THEN
				sState 				:=	'Undefined' ;
	ELSIF stInfoData.usiMapState 	= 	2 THEN
				sState 				:= 	'STOP' ;
	ELSIF stInfoData.usiMapState 	= 	3 THEN
				sState 				:= 	'SAFE' ;
	ELSIF stInfoData.usiMapState 	= 	4 THEN
				sState 				:= 	'Error' ;
	ELSIF stInfoData.usiMapState 	= 	5 THEN
				sState 				:= 	'Reset' ;
	ELSIF stInfoData.usiMapState 	= 	10 THEN
				sState 				:= 	'Active' ;
	ELSIF stInfoData.usiMapState 	= 	11 THEN
				sState 				:= 	'Deactive' ;
	ELSE
				sState 				:= 	'Unknown' ;
END_IF

// Connection Shutdown FB's Diagnostics
IF stInfoData.uiMapDiag 			= 	0 THEN
				sDiag 				:= 	'No Error' ;
ELSIF  stInfoData.uiMapDiag 		= 	1 THEN
				sDiag 				:= 	'Discrepancy Error Input Group1' ;
ELSE
				sDiag 				:= 	'Unknown' ;
END_IF

END_FUNCTION_BLOCK

// ---- POUs/TwinSAFE_Function_Blocks_Info/FB_InfoOR.TcPOU
FUNCTION_BLOCK FB_InfoOR
VAR_INPUT
	stInfoData 			: 		DUT_ST_InfoDataFB ;
END_VAR
VAR_OUTPUT
	sState 				: 		STRING ;
END_VAR
VAR
END_VAR

// OR FB's State
IF stInfoData.usiMapState 			= 	0 THEN
				sState 				:= 	'Undefined' ;
	ELSIF stInfoData.usiMapState 	= 	1 THEN
				sState 				:= 	'RUN' ;
	ELSIF stInfoData.usiMapState 	= 	2 THEN
				sState 				:= 	'STOP' ;
	ELSIF stInfoData.usiMapState 	= 	3 THEN
				sState 				:= 	'SAFE' ;
	ELSE
				sState 				:= 	'Unknown' ;
END_IF

// The OR FB Has No Diagnostic Byte to Decode

END_FUNCTION_BLOCK

